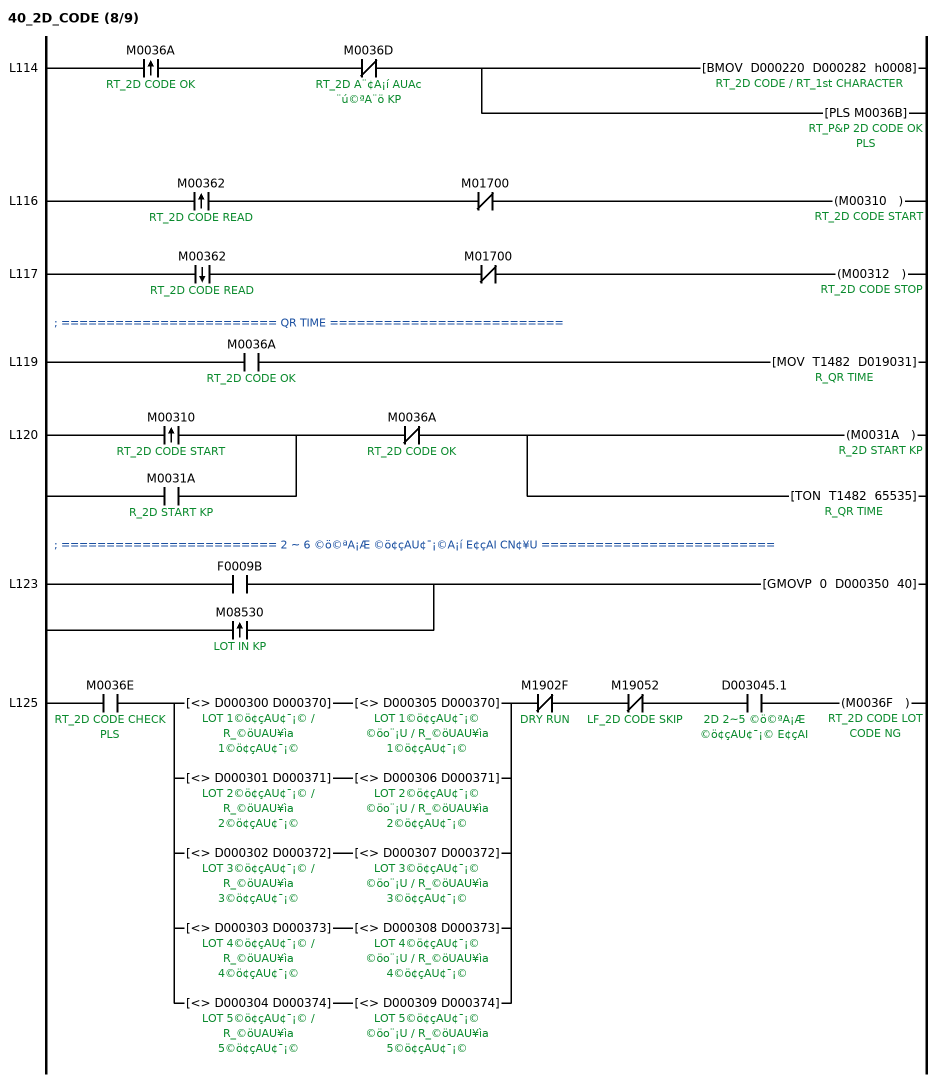
[picture p240: 40_2D_CODE rungs L114-L125]
; L114
LOADP     M0036A	// RT_2D CODE OK
AND NOT   M0036D	// RT_2D A¨¢A¡í AUAc ¨ú©ªA¨ö KP
BMOV      D000220 D000282 h0008	// RT_2D CODE / RT_1st CHARACTER
OUTP      M0036B	// RT_P&P 2D CODE OK PLS
; L116
LOADP     M00362	// RT_2D CODE READ
AND NOT   M01700
OUT       M00310	// RT_2D CODE START
; L117
LOADN     M00362	// RT_2D CODE READ
AND NOT   M01700
OUT       M00312	// RT_2D CODE STOP
// ======================== QR TIME ==========================
; L119
LOAD      M0036A	// RT_2D CODE OK
MOV       T1482 D019031	// R_QR TIME
; L120
LOADP     M00310	// RT_2D CODE START
OR        M0031A	// R_2D START KP
AND NOT   M0036A	// RT_2D CODE OK
OUT       M0031A	// R_2D START KP
TON       T1482 65535	// R_QR TIME
// ======================== 2 ~ 6 ©ö©ªA¡Æ ©ö¢çAU¢¯¡©A¡í E¢çAI CN¢¥U ==========================
; L123
LOAD      F0009B
ORP       M08530	// LOT IN KP
GMOVP     0 D000350 40
; L125
LOAD      M0036E	// RT_2D CODE CHECK PLS
LOAD<>    D000300 D000370	// LOT 1©ö¢çAU¢¯¡© / R_©öUAU¥ìa 1©ö¢çAU¢¯¡©
AND<>     D000305 D000370	// LOT 1©ö¢çAU¢¯¡© ©öo¨¡U / R_©öUAU¥ìa 1©ö¢çAU¢¯¡©
LOAD<>    D000301 D000371	// LOT 2©ö¢çAU¢¯¡© / R_©öUAU¥ìa 2©ö¢çAU¢¯¡©
AND<>     D000306 D000371	// LOT 2©ö¢çAU¢¯¡© ©öo¨¡U / R_©öUAU¥ìa 2©ö¢çAU¢¯¡©
OR LOAD
LOAD<>    D000302 D000372	// LOT 3©ö¢çAU¢¯¡© / R_©öUAU¥ìa 3©ö¢çAU¢¯¡©
AND<>     D000307 D000372	// LOT 3©ö¢çAU¢¯¡© ©öo¨¡U / R_©öUAU¥ìa 3©ö¢çAU¢¯¡©
OR LOAD
LOAD<>    D000303 D000373	// LOT 4©ö¢çAU¢¯¡© / R_©öUAU¥ìa 4©ö¢çAU¢¯¡©
AND<>     D000308 D000373	// LOT 4©ö¢çAU¢¯¡© ©öo¨¡U / R_©öUAU¥ìa 4©ö¢çAU¢¯¡©
OR LOAD
LOAD<>    D000304 D000374	// LOT 5©ö¢çAU¢¯¡© / R_©öUAU¥ìa 5©ö¢çAU¢¯¡©
AND<>     D000309 D000374	// LOT 5©ö¢çAU¢¯¡© ©öo¨¡U / R_©öUAU¥ìa 5©ö¢çAU¢¯¡©
OR LOAD
AND LOAD
AND NOT   M1902F	// DRY RUN
AND NOT   M19052	// LF_2D CODE SKIP
AND       D003045.1	// 2D 2~5 ©ö©ªA¡Æ ©ö¢çAU¢¯¡© E¢çAI
OUT       M0036F	// RT_2D CODE LOT CODE NG

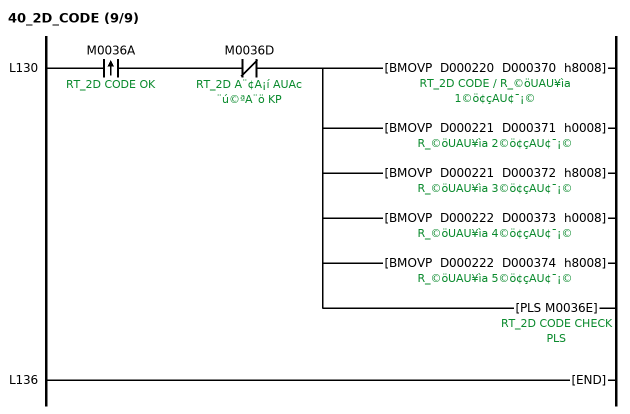
; L130
LOADP     M0036A	// RT_2D CODE OK
AND NOT   M0036D	// RT_2D A¨¢A¡í AUAc ¨ú©ªA¨ö KP
BMOVP     D000220 D000370 h8008	// RT_2D CODE / R_©öUAU¥ìa 1©ö¢çAU¢¯¡©
BMOVP     D000221 D000371 h0008	// R_©öUAU¥ìa 2©ö¢çAU¢¯¡©
BMOVP     D000221 D000372 h8008	// R_©öUAU¥ìa 3©ö¢çAU¢¯¡©
BMOVP     D000222 D000373 h0008	// R_©öUAU¥ìa 4©ö¢çAU¢¯¡©
BMOVP     D000222 D000374 h8008	// R_©öUAU¥ìa 5©ö¢çAU¢¯¡©
OUTP      M0036E	// RT_2D CODE CHECK PLS
; L136
END

PROGRAM 41_MES (task: ¨ö¨¬A¥ì CA¡¤I¡¾¡¿¡¤¡Í)

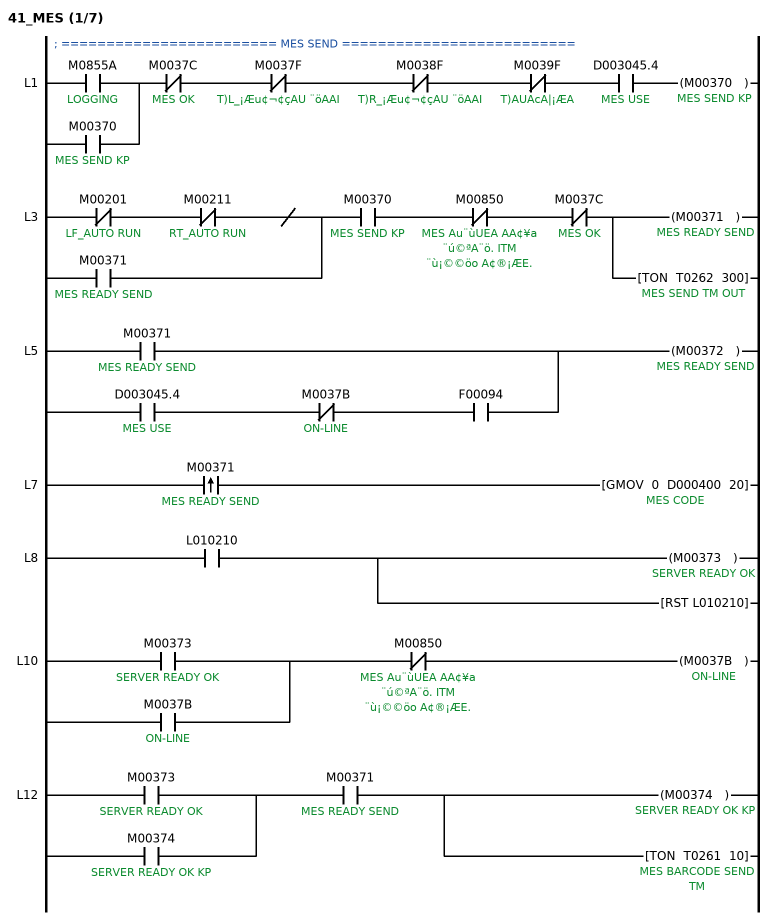
// ======================== MES SEND ==========================
; L1
LOAD      M0855A	// LOGGING
OR        M00370	// MES SEND KP
AND NOT   M0037C	// MES OK
AND NOT   M0037F	// T)L_¡Æu¢¬¢çAU ¨öAAI
AND NOT   M0038F	// T)R_¡Æu¢¬¢çAU ¨öAAI
AND NOT   M0039F	// T)AUAcA|¡ÆA
AND       D003045.4	// MES USE
OUT       M00370	// MES SEND KP
; L3
LOAD NOT  M00201	// LF_AUTO RUN
AND NOT   M00211	// RT_AUTO RUN
NOT
OR        M00371	// MES READY SEND
AND       M00370	// MES SEND KP
AND NOT   M00850	// MES Au¨ùUEA AA¢¥a ¨ú©ªA¨ö. ITM ¨ù¡©©öo A¢®¡ÆE.
AND NOT   M0037C	// MES OK
OUT       M00371	// MES READY SEND
TON       T0262 300	// MES SEND TM OUT
; L5
LOAD      M00371	// MES READY SEND
LOAD      D003045.4	// MES USE
AND NOT   M0037B	// ON-LINE
AND       F00094
OR LOAD
OUT       M00372	// MES READY SEND
; L7
LOADP     M00371	// MES READY SEND
GMOV      0 D000400 20	// MES CODE
; L8
LOAD      L010210
OUT       M00373	// SERVER READY OK
RST       L010210
; L10
LOAD      M00373	// SERVER READY OK
OR        M0037B	// ON-LINE
AND NOT   M00850	// MES Au¨ùUEA AA¢¥a ¨ú©ªA¨ö. ITM ¨ù¡©©öo A¢®¡ÆE.
OUT       M0037B	// ON-LINE
; L12
LOAD      M00373	// SERVER READY OK
OR        M00374	// SERVER READY OK KP
AND       M00371	// MES READY SEND
OUT       M00374	// SERVER READY OK KP
TON       T0261 10	// MES BARCODE SEND TM

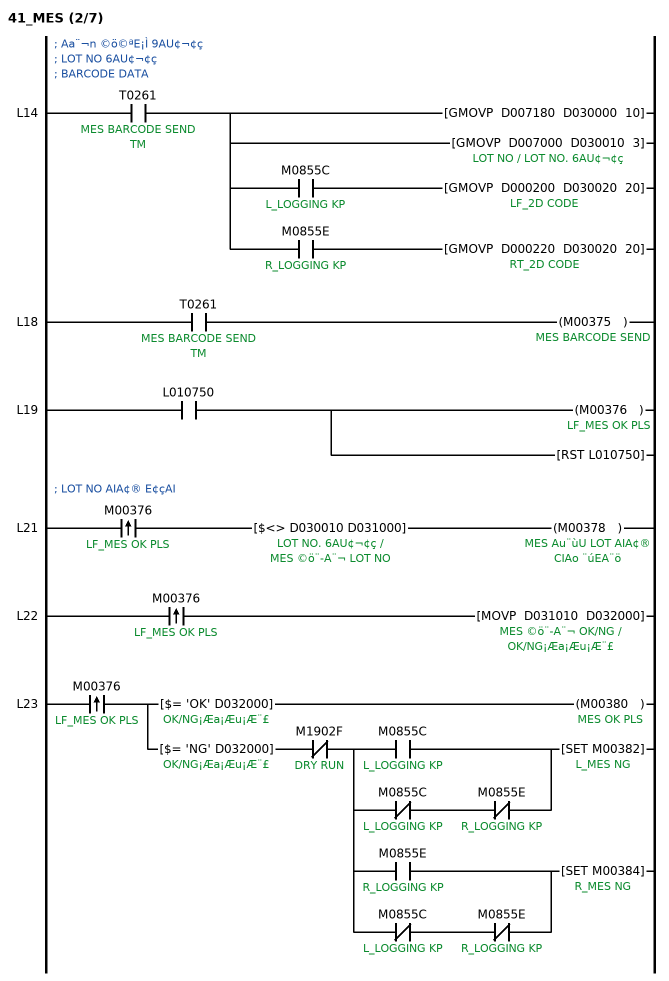
; L14
LOAD      T0261	// MES BARCODE SEND TM
GMOVP     D007180 D030000 10
GMOVP     D007000 D030010 3	// LOT NO / LOT NO. 6AU¢¬¢ç
MPUSH
AND       M0855C	// L_LOGGING KP
GMOVP     D000200 D030020 20	// LF_2D CODE
MPOP
AND       M0855E	// R_LOGGING KP
GMOVP     D000220 D030020 20	// RT_2D CODE
// output comment: Aa¨¬n ©ö©ªE¡Ì 9AU¢¬¢ç
// output comment: LOT NO 6AU¢¬¢ç
// output comment: BARCODE DATA
; L18
LOAD      T0261	// MES BARCODE SEND TM
OUT       M00375	// MES BARCODE SEND
; L19
LOAD      L010750
OUT       M00376	// LF_MES OK PLS
RST       L010750
; L21
LOADP     M00376	// LF_MES OK PLS
AND$<>    D030010 D031000	// LOT NO. 6AU¢¬¢ç / MES ©ö¨­A¨¬ LOT NO
OUT       M00378	// MES Au¨ùU LOT AIA¢® CIAo ¨úEA¨ö
// output comment: LOT NO AIA¢® E¢çAI
; L22
LOADP     M00376	// LF_MES OK PLS
MOVP      D031010 D032000	// MES ©ö¨­A¨¬ OK/NG / OK/NG¡Æa¡Æu¡Æ¨£
; L23
LOADP     M00376	// LF_MES OK PLS
MPUSH
AND$=     'OK' D032000	// OK/NG¡Æa¡Æu¡Æ¨£
OUT       M00380	// MES OK PLS
MPOP
AND$=     'NG' D032000	// OK/NG¡Æa¡Æu¡Æ¨£
AND NOT   M1902F	// DRY RUN
MPUSH
LOAD      M0855C	// L_LOGGING KP
LOAD NOT  M0855C	// L_LOGGING KP
AND NOT   M0855E	// R_LOGGING KP
OR LOAD
AND LOAD
SET       M00382	// L_MES NG
MPOP
LOAD      M0855E	// R_LOGGING KP
LOAD NOT  M0855C	// L_LOGGING KP
AND NOT   M0855E	// R_LOGGING KP
OR LOAD
AND LOAD
SET       M00384	// R_MES NG

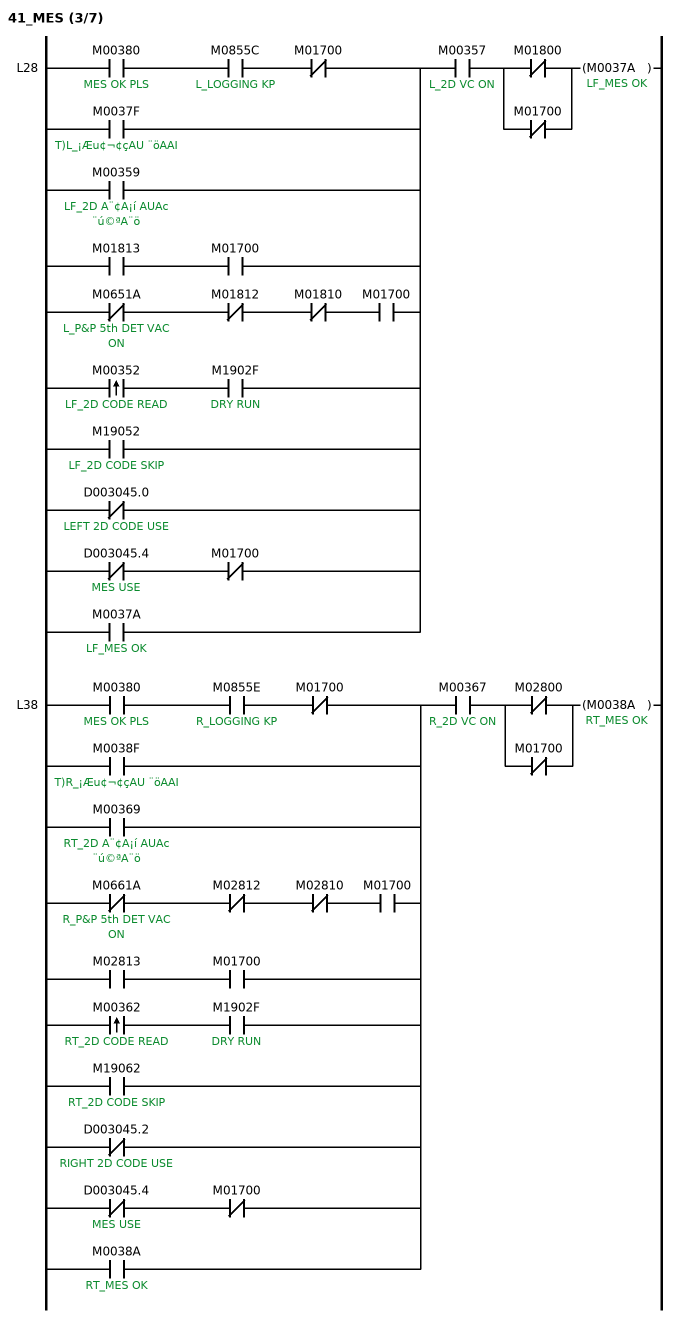
; L28
LOAD      M00380	// MES OK PLS
AND       M0855C	// L_LOGGING KP
AND NOT   M01700
OR        M0037F	// T)L_¡Æu¢¬¢çAU ¨öAAI
OR        M00359	// LF_2D A¨¢A¡í AUAc ¨ú©ªA¨ö
LOAD      M01813
AND       M01700
OR LOAD
LOAD NOT  M0651A	// L_P&P 5th DET VAC ON
AND NOT   M01812
AND NOT   M01810
AND       M01700
OR LOAD
LOADP     M00352	// LF_2D CODE READ
AND       M1902F	// DRY RUN
OR LOAD
OR        M19052	// LF_2D CODE SKIP
OR NOT    D003045.0	// LEFT 2D CODE USE
LOAD NOT  D003045.4	// MES USE
AND NOT   M01700
OR LOAD
OR        M0037A	// LF_MES OK
AND       M00357	// L_2D VC ON
LOAD NOT  M01800
OR NOT    M01700
AND LOAD
OUT       M0037A	// LF_MES OK
; L38
LOAD      M00380	// MES OK PLS
AND       M0855E	// R_LOGGING KP
AND NOT   M01700
OR        M0038F	// T)R_¡Æu¢¬¢çAU ¨öAAI
OR        M00369	// RT_2D A¨¢A¡í AUAc ¨ú©ªA¨ö
LOAD NOT  M0661A	// R_P&P 5th DET VAC ON
AND NOT   M02812
AND NOT   M02810
AND       M01700
OR LOAD
LOAD      M02813
AND       M01700
OR LOAD
LOADP     M00362	// RT_2D CODE READ
AND       M1902F	// DRY RUN
OR LOAD
OR        M19062	// RT_2D CODE SKIP
OR NOT    D003045.2	// RIGHT 2D CODE USE
LOAD NOT  D003045.4	// MES USE
AND NOT   M01700
OR LOAD
OR        M0038A	// RT_MES OK
AND       M00367	// R_2D VC ON
LOAD NOT  M02800
OR NOT    M01700
AND LOAD
OUT       M0038A	// RT_MES OK

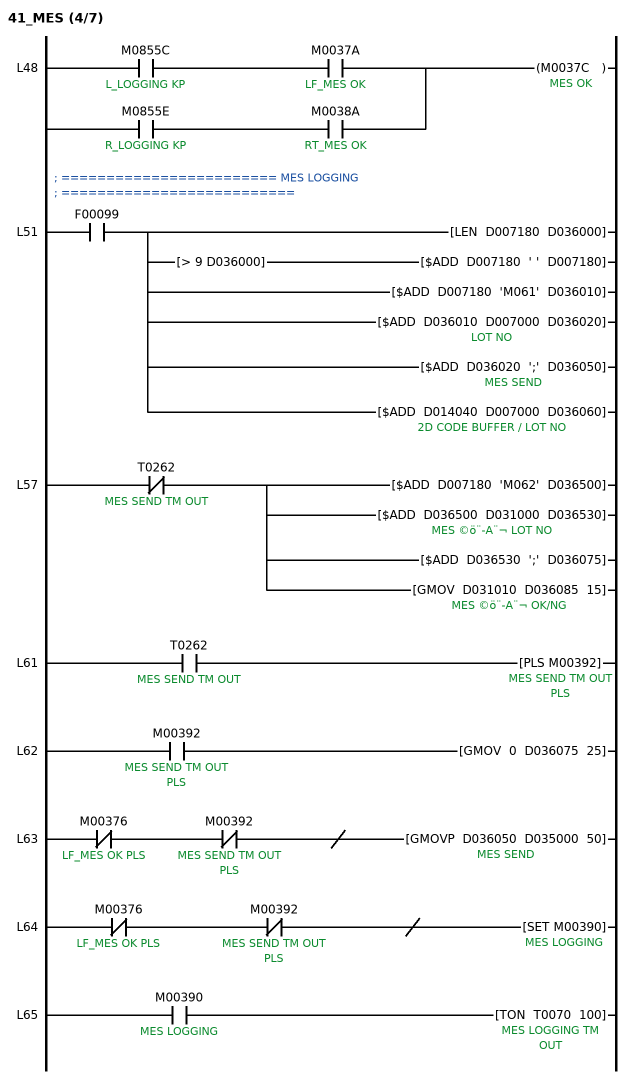
; L48
LOAD      M0855C	// L_LOGGING KP
AND       M0037A	// LF_MES OK
LOAD      M0855E	// R_LOGGING KP
AND       M0038A	// RT_MES OK
OR LOAD
OUT       M0037C	// MES OK
// ======================== MES LOGGING ==========================
; L51
LOAD      F00099
LEN       D007180 D036000
MPUSH
AND>      9 D036000
$ADD      D007180 ' ' D007180
MPOP
$ADD      D007180 'M061' D036010
$ADD      D036010 D007000 D036020	// LOT NO
$ADD      D036020 ';' D036050	// MES SEND
$ADD      D014040 D007000 D036060	// 2D CODE BUFFER / LOT NO
; L57
LOAD NOT  T0262	// MES SEND TM OUT
$ADD      D007180 'M062' D036500
$ADD      D036500 D031000 D036530	// MES ©ö¨­A¨¬ LOT NO
$ADD      D036530 ';' D036075
GMOV      D031010 D036085 15	// MES ©ö¨­A¨¬ OK/NG
; L61
LOAD      T0262	// MES SEND TM OUT
OUTP      M00392	// MES SEND TM OUT PLS
; L62
LOAD      M00392	// MES SEND TM OUT PLS
GMOV      0 D036075 25
; L63
LOAD NOT  M00376	// LF_MES OK PLS
AND NOT   M00392	// MES SEND TM OUT PLS
NOT
GMOVP     D036050 D035000 50	// MES SEND
; L64
LOAD NOT  M00376	// LF_MES OK PLS
AND NOT   M00392	// MES SEND TM OUT PLS
NOT
SET       M00390	// MES LOGGING
; L65
LOAD      M00390	// MES LOGGING
TON       T0070 100	// MES LOGGING TM OUT

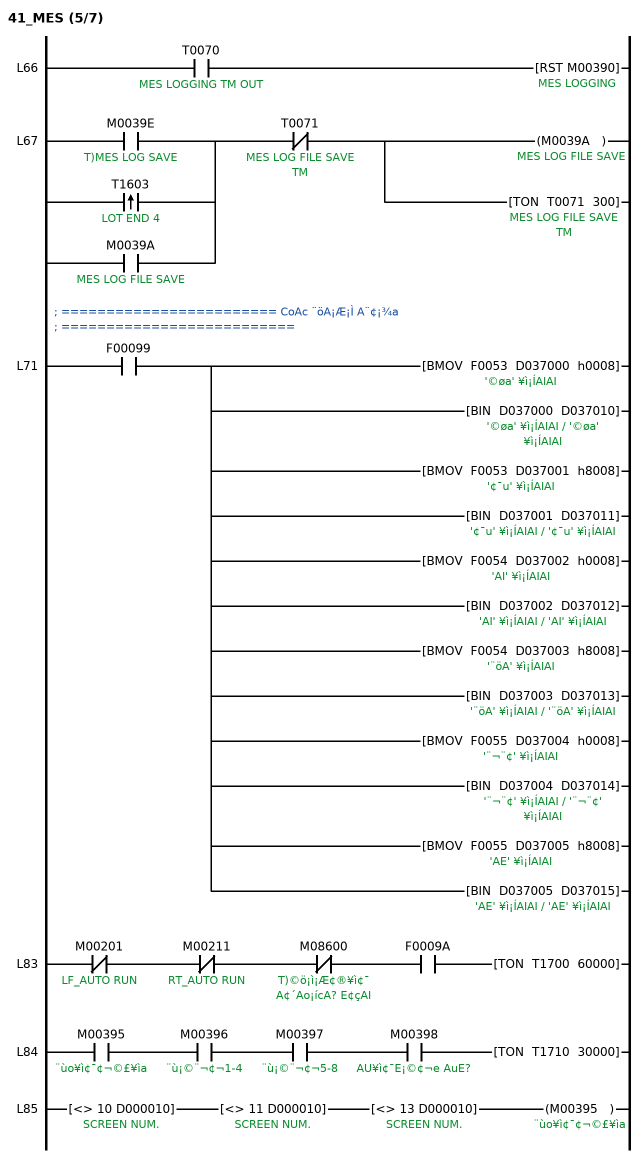
; L66
LOAD      T0070	// MES LOGGING TM OUT
RST       M00390	// MES LOGGING
; L67
LOAD      M0039E	// T)MES LOG SAVE
ORP       T1603	// LOT END 4
OR        M0039A	// MES LOG FILE SAVE
AND NOT   T0071	// MES LOG FILE SAVE TM
OUT       M0039A	// MES LOG FILE SAVE
TON       T0071 300	// MES LOG FILE SAVE TM
// ======================== CoAc ¨öA¡Æ¡Ì A¨¢¡¾a ==========================
; L71
LOAD      F00099
BMOV      F0053 D037000 h0008	// '©øa' ¥ì¡ÍAIAI
BIN       D037000 D037010	// '©øa' ¥ì¡ÍAIAI / '©øa' ¥ì¡ÍAIAI
BMOV      F0053 D037001 h8008	// '¢¯u' ¥ì¡ÍAIAI
BIN       D037001 D037011	// '¢¯u' ¥ì¡ÍAIAI / '¢¯u' ¥ì¡ÍAIAI
BMOV      F0054 D037002 h0008	// 'AI' ¥ì¡ÍAIAI
BIN       D037002 D037012	// 'AI' ¥ì¡ÍAIAI / 'AI' ¥ì¡ÍAIAI
BMOV      F0054 D037003 h8008	// '¨öA' ¥ì¡ÍAIAI
BIN       D037003 D037013	// '¨öA' ¥ì¡ÍAIAI / '¨öA' ¥ì¡ÍAIAI
BMOV      F0055 D037004 h0008	// '¨¬¨¢' ¥ì¡ÍAIAI
BIN       D037004 D037014	// '¨¬¨¢' ¥ì¡ÍAIAI / '¨¬¨¢' ¥ì¡ÍAIAI
BMOV      F0055 D037005 h8008	// 'AE' ¥ì¡ÍAIAI
BIN       D037005 D037015	// 'AE' ¥ì¡ÍAIAI / 'AE' ¥ì¡ÍAIAI
; L83
LOAD NOT  M00201	// LF_AUTO RUN
AND NOT   M00211	// RT_AUTO RUN
AND NOT   M08600	// T)©ö¡ì¡Æ¢®¥ì¢¯ A¢´Ao¡ícA? E¢çAI
AND       F0009A
TON       T1700 60000
; L84
LOAD      M00395	// ¨ùo¥ì¢¯¢¬©£¥ìa
AND       M00396	// ¨ù¡©¨¬¢¬1-4
AND       M00397	// ¨ù¡©¨¬¢¬5-8
AND       M00398	// AU¥ì¢¯E¡©¢¬e AuE?
TON       T1710 30000
; L85
LOAD<>    10 D000010	// SCREEN NUM.
AND<>     11 D000010	// SCREEN NUM.
AND<>     13 D000010	// SCREEN NUM.
OUT       M00395	// ¨ùo¥ì¢¯¢¬©£¥ìa

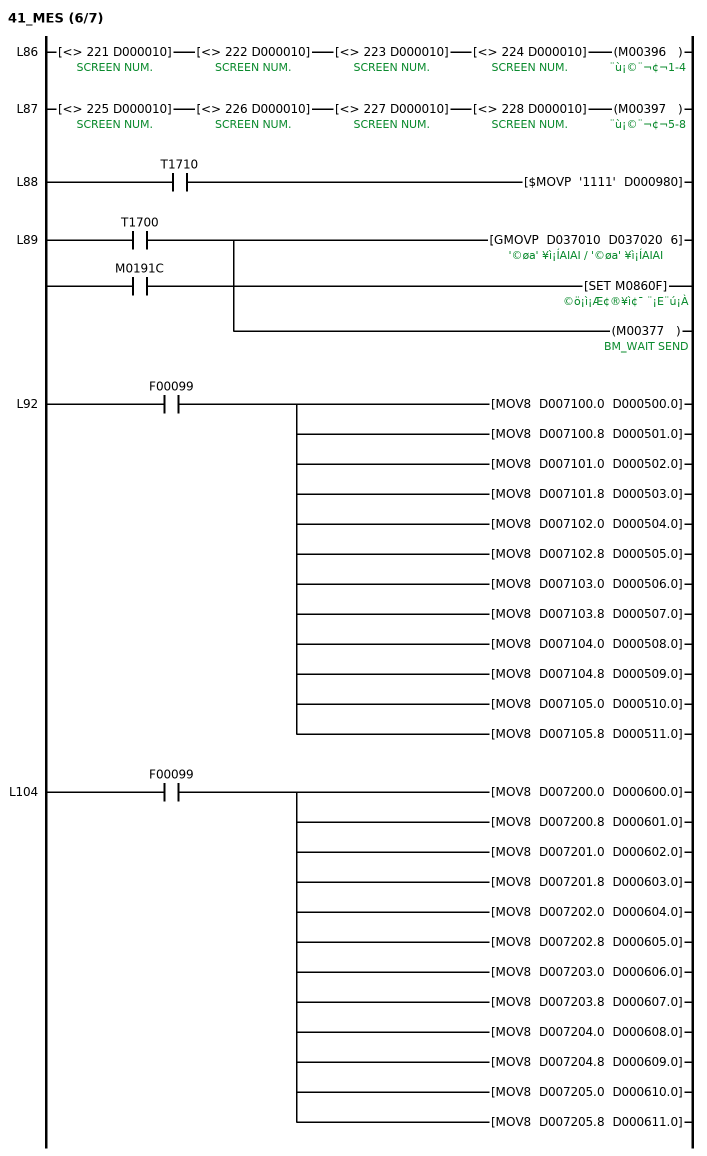
; L86
LOAD<>    221 D000010	// SCREEN NUM.
AND<>     222 D000010	// SCREEN NUM.
AND<>     223 D000010	// SCREEN NUM.
AND<>     224 D000010	// SCREEN NUM.
OUT       M00396	// ¨ù¡©¨¬¢¬1-4
; L87
LOAD<>    225 D000010	// SCREEN NUM.
AND<>     226 D000010	// SCREEN NUM.
AND<>     227 D000010	// SCREEN NUM.
AND<>     228 D000010	// SCREEN NUM.
OUT       M00397	// ¨ù¡©¨¬¢¬5-8
; L88
LOAD      T1710
$MOVP     '1111' D000980
; L89
LOAD      T1700
OR        M0191C
GMOVP     D037010 D037020 6	// '©øa' ¥ì¡ÍAIAI / '©øa' ¥ì¡ÍAIAI
SET       M0860F	// ©ö¡ì¡Æ¢®¥ì¢¯ ¨¡E¨ú¡À
OUT       M00377	// BM_WAIT SEND
; L92
LOAD      F00099
MOV8      D007100.0 D000500.0
MOV8      D007100.8 D000501.0
MOV8      D007101.0 D000502.0
MOV8      D007101.8 D000503.0
MOV8      D007102.0 D000504.0
MOV8      D007102.8 D000505.0
MOV8      D007103.0 D000506.0
MOV8      D007103.8 D000507.0
MOV8      D007104.0 D000508.0
MOV8      D007104.8 D000509.0
MOV8      D007105.0 D000510.0
MOV8      D007105.8 D000511.0
; L104
LOAD      F00099
MOV8      D007200.0 D000600.0
MOV8      D007200.8 D000601.0
MOV8      D007201.0 D000602.0
MOV8      D007201.8 D000603.0
MOV8      D007202.0 D000604.0
MOV8      D007202.8 D000605.0
MOV8      D007203.0 D000606.0
MOV8      D007203.8 D000607.0
MOV8      D007204.0 D000608.0
MOV8      D007204.8 D000609.0
MOV8      D007205.0 D000610.0
MOV8      D007205.8 D000611.0

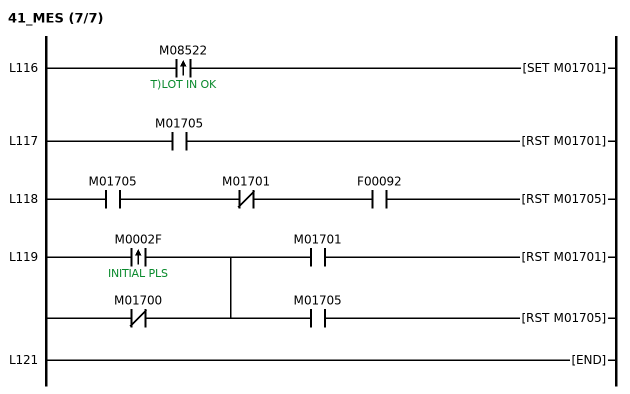
; L116
LOADP     M08522	// T)LOT IN OK
SET       M01701
; L117
LOAD      M01705
RST       M01701
; L118
LOAD      M01705
AND NOT   M01701
AND       F00092
RST       M01705
; L119
LOADP     M0002F	// INITIAL PLS
OR NOT    M01700
MPUSH
AND       M01701
RST       M01701
MPOP
AND       M01705
RST       M01705
; L121
END

PROGRAM 51_MT_01_2_3_4 (task: ¨ö¨¬A¥ì CA¡¤I¡¾¡¿¡¤¡Í)

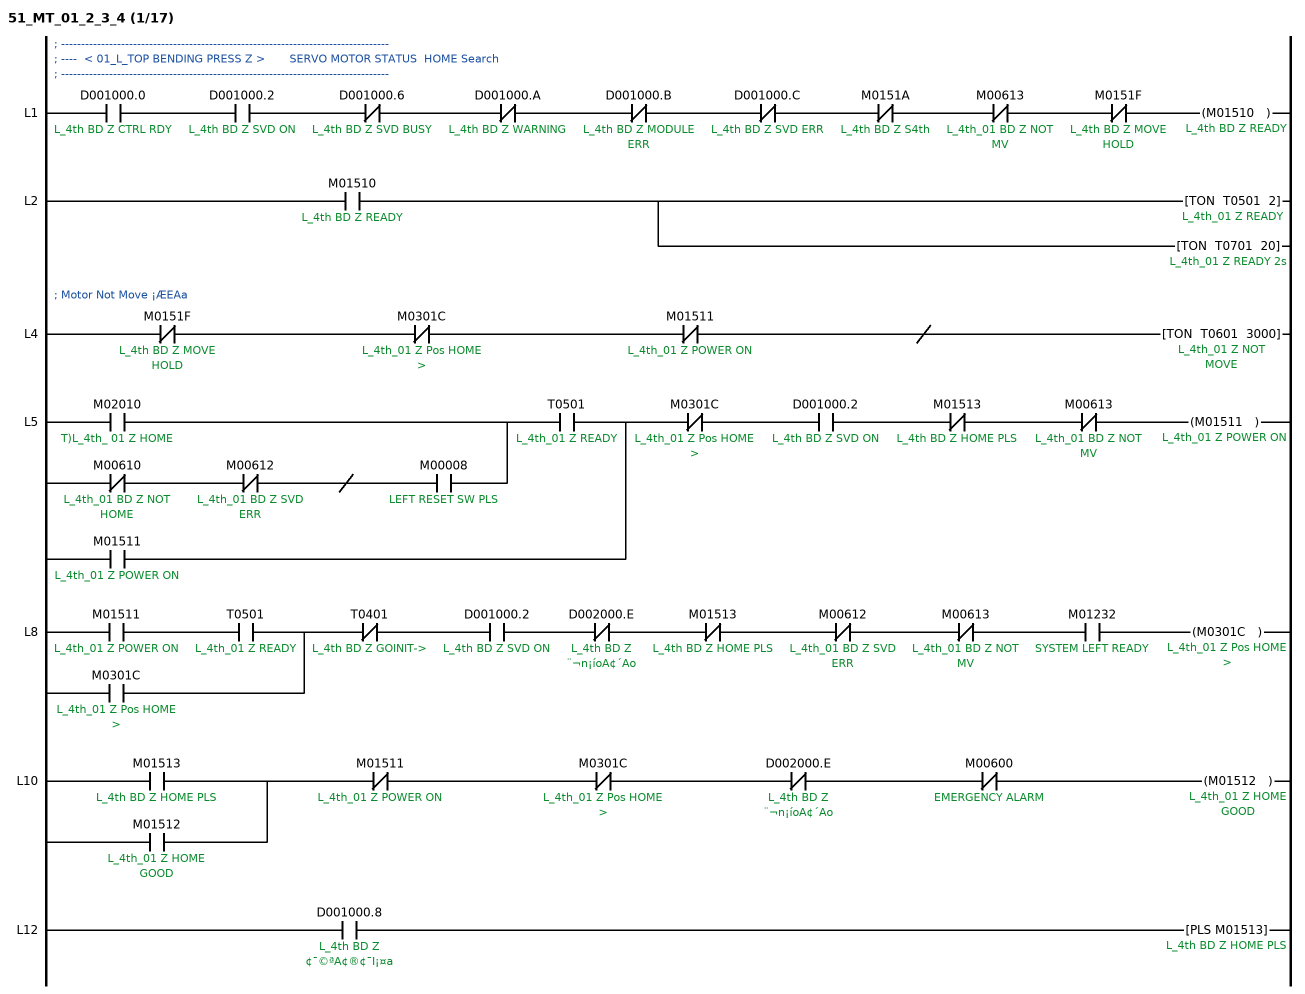
// ----------------------------------------------------------------------------------
// 
// ----  < 01_L_TOP BENDING PRESS Z >       SERVO MOTOR STATUS  HOME Search
// 
// ----------------------------------------------------------------------------------
; L1
LOAD      D001000.0	// L_4th BD Z CTRL RDY
AND       D001000.2	// L_4th BD Z SVD ON
AND NOT   D001000.6	// L_4th BD Z SVD BUSY
AND NOT   D001000.A	// L_4th BD Z WARNING
AND NOT   D001000.B	// L_4th BD Z MODULE ERR
AND NOT   D001000.C	// L_4th BD Z SVD ERR
AND NOT   M0151A	// L_4th BD Z S4th
AND NOT   M00613	// L_4th_01 BD Z NOT MV
AND NOT   M0151F	// L_4th BD Z MOVE HOLD
OUT       M01510	// L_4th BD Z READY
; L2
LOAD      M01510	// L_4th BD Z READY
TON       T0501 2	// L_4th_01 Z READY
TON       T0701 20	// L_4th_01 Z READY 2s
; L4
LOAD NOT  M0151F	// L_4th BD Z MOVE HOLD
AND NOT   M0301C	// L_4th_01 Z Pos HOME >
AND NOT   M01511	// L_4th_01 Z POWER ON
NOT
TON       T0601 3000	// L_4th_01 Z NOT MOVE
// output comment: Motor Not Move ¡ÆEAa
; L5
LOAD      M02010	// T)L_4th_ 01 Z HOME
LOAD NOT  M00610	// L_4th_01 BD Z NOT HOME
AND NOT   M00612	// L_4th_01 BD Z SVD ERR
NOT
AND       M00008	// LEFT RESET SW PLS
OR LOAD
AND       T0501	// L_4th_01 Z READY
OR        M01511	// L_4th_01 Z POWER ON
AND NOT   M0301C	// L_4th_01 Z Pos HOME >
AND       D001000.2	// L_4th BD Z SVD ON
AND NOT   M01513	// L_4th BD Z HOME PLS
AND NOT   M00613	// L_4th_01 BD Z NOT MV
OUT       M01511	// L_4th_01 Z POWER ON
; L8
LOAD      M01511	// L_4th_01 Z POWER ON
AND       T0501	// L_4th_01 Z READY
OR        M0301C	// L_4th_01 Z Pos HOME >
AND NOT   T0401	// L_4th BD Z GOINIT->
AND       D001000.2	// L_4th BD Z SVD ON
AND NOT   D002000.E	// L_4th BD Z ¨¬n¡íoA¢´Ao
AND NOT   M01513	// L_4th BD Z HOME PLS
AND NOT   M00612	// L_4th_01 BD Z SVD ERR
AND NOT   M00613	// L_4th_01 BD Z NOT MV
AND       M01232	// SYSTEM LEFT READY
OUT       M0301C	// L_4th_01 Z Pos HOME >
; L10
LOAD      M01513	// L_4th BD Z HOME PLS
OR        M01512	// L_4th_01 Z HOME GOOD
AND NOT   M01511	// L_4th_01 Z POWER ON
AND NOT   M0301C	// L_4th_01 Z Pos HOME >
AND NOT   D002000.E	// L_4th BD Z ¨¬n¡íoA¢´Ao
AND NOT   M00600	// EMERGENCY ALARM
OUT       M01512	// L_4th_01 Z HOME GOOD
; L12
LOAD      D001000.8	// L_4th BD Z ¢¯©ªA¢®¢¯I¡¤a
OUTP      M01513	// L_4th BD Z HOME PLS

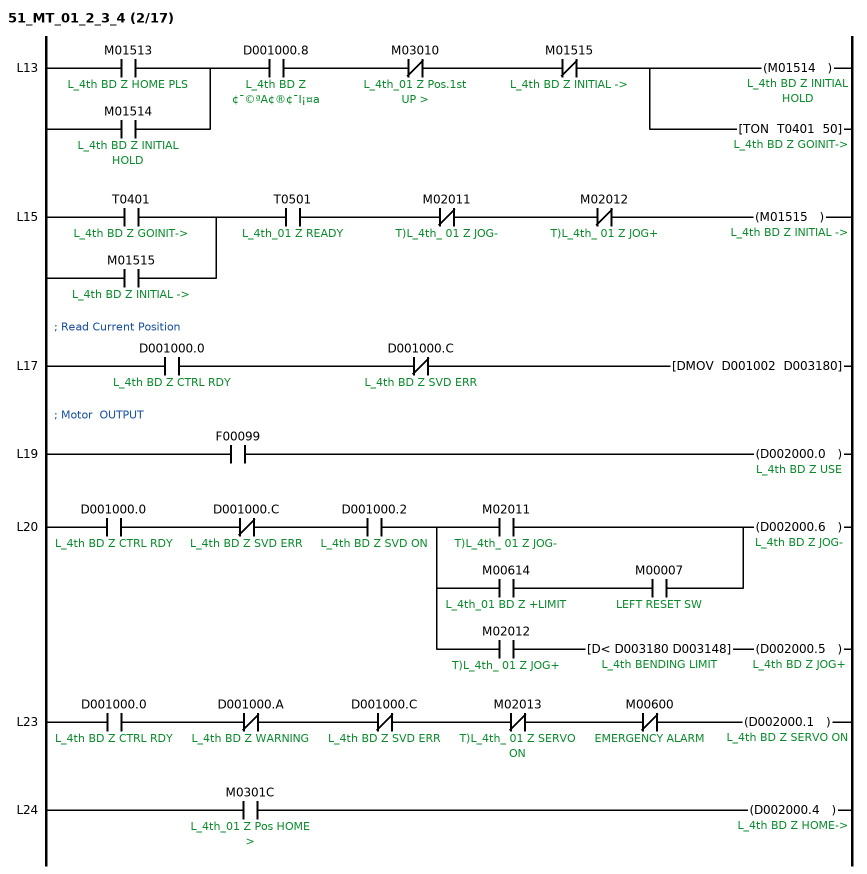
; L13
LOAD      M01513	// L_4th BD Z HOME PLS
OR        M01514	// L_4th BD Z INITIAL HOLD
AND       D001000.8	// L_4th BD Z ¢¯©ªA¢®¢¯I¡¤a
AND NOT   M03010	// L_4th_01 Z Pos.1st     UP >
AND NOT   M01515	// L_4th BD Z INITIAL ->
OUT       M01514	// L_4th BD Z INITIAL HOLD
TON       T0401 50	// L_4th BD Z GOINIT->
; L15
LOAD      T0401	// L_4th BD Z GOINIT->
OR        M01515	// L_4th BD Z INITIAL ->
AND       T0501	// L_4th_01 Z READY
AND NOT   M02011	// T)L_4th_ 01 Z JOG-
AND NOT   M02012	// T)L_4th_ 01 Z JOG+
OUT       M01515	// L_4th BD Z INITIAL ->
; L17
LOAD      D001000.0	// L_4th BD Z CTRL RDY
AND NOT   D001000.C	// L_4th BD Z SVD ERR
DMOV      D001002 D003180
// output comment: Read Current Position
//  Motor  OUTPUT
; L19
LOAD      F00099
OUT       D002000.0	// L_4th BD Z USE
; L20
LOAD      D001000.0	// L_4th BD Z CTRL RDY
AND NOT   D001000.C	// L_4th BD Z SVD ERR
AND       D001000.2	// L_4th BD Z SVD ON
MPUSH
LOAD      M02011	// T)L_4th_ 01 Z JOG-
LOAD      M00614	// L_4th_01 BD Z +LIMIT
AND       M00007	// LEFT RESET SW
OR LOAD
AND LOAD
OUT       D002000.6	// L_4th BD Z JOG-
MPOP
AND       M02012	// T)L_4th_ 01 Z JOG+
ANDD<     D003180 D003148	// L_4th BENDING LIMIT
OUT       D002000.5	// L_4th BD Z JOG+
; L23
LOAD      D001000.0	// L_4th BD Z CTRL RDY
AND NOT   D001000.A	// L_4th BD Z WARNING
AND NOT   D001000.C	// L_4th BD Z SVD ERR
AND NOT   M02013	// T)L_4th_ 01 Z SERVO ON
AND NOT   M00600	// EMERGENCY ALARM
OUT       D002000.1	// L_4th BD Z SERVO ON
; L24
LOAD      M0301C	// L_4th_01 Z Pos HOME >
OUT       D002000.4	// L_4th BD Z HOME->

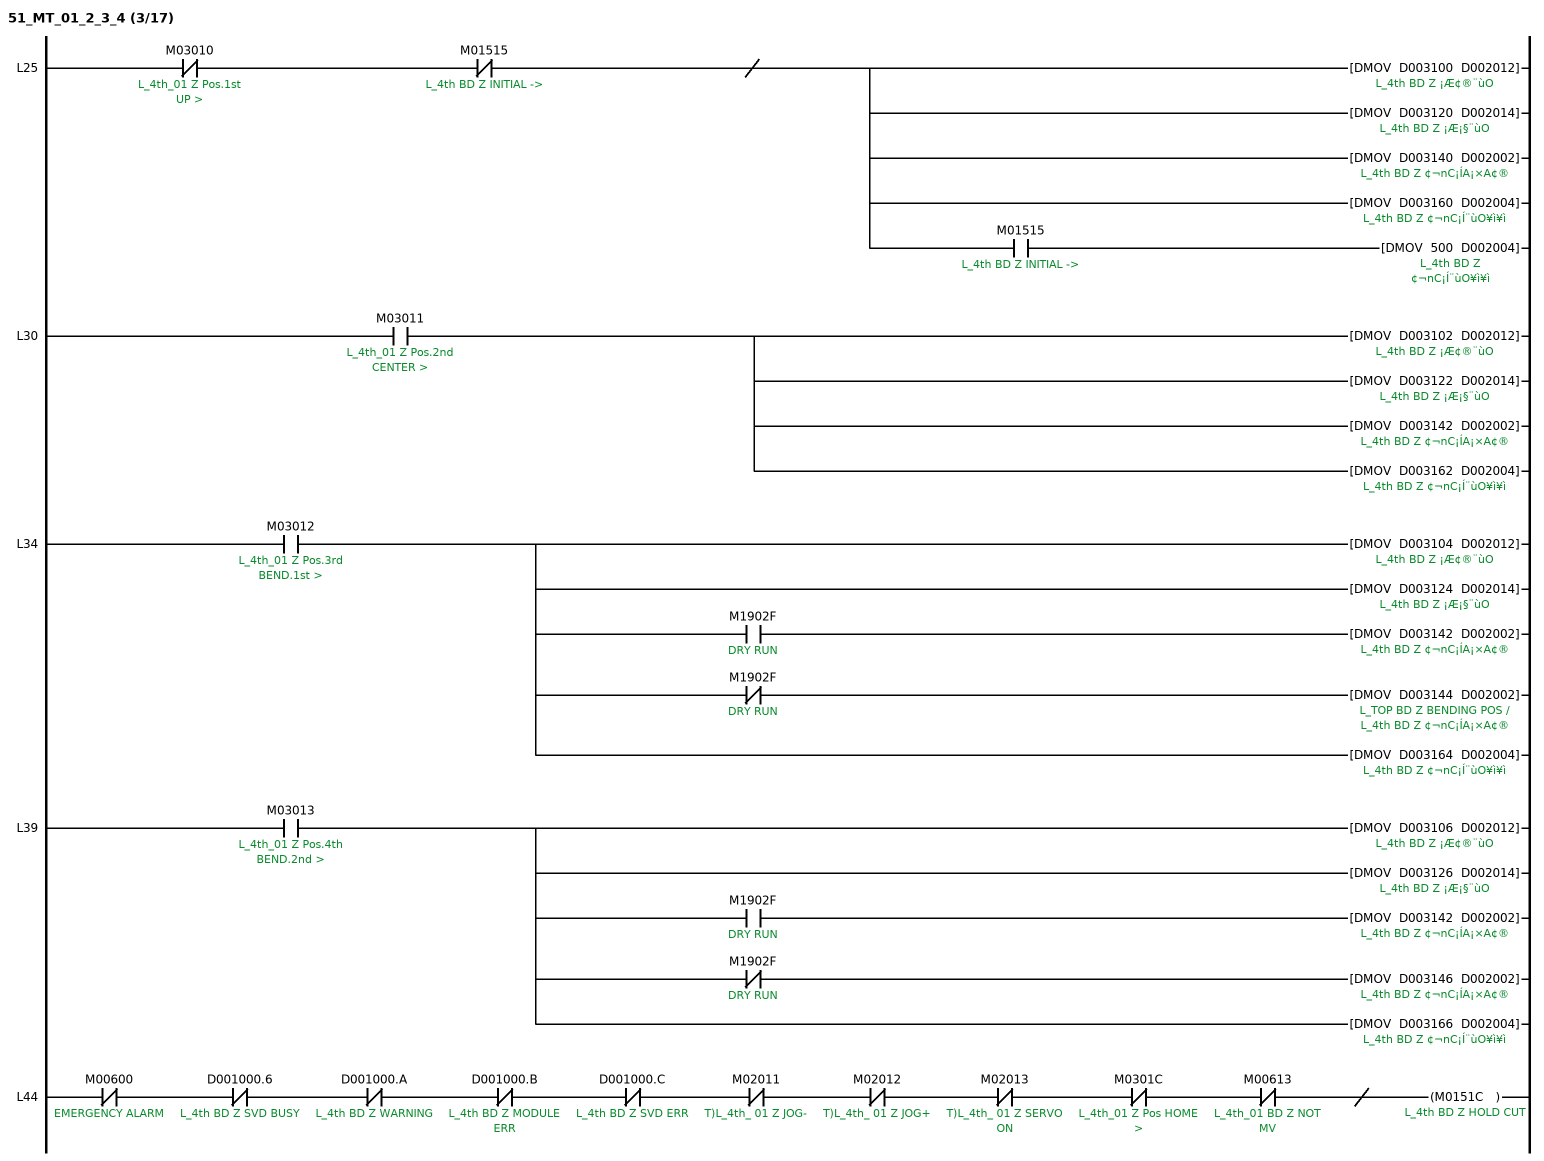
; L25
LOAD NOT  M03010	// L_4th_01 Z Pos.1st     UP >
AND NOT   M01515	// L_4th BD Z INITIAL ->
NOT
DMOV      D003100 D002012	// L_4th BD Z ¡Æ¢®¨ùO
DMOV      D003120 D002014	// L_4th BD Z ¡Æ¡§¨ùO
DMOV      D003140 D002002	// L_4th BD Z ¢¬nC¡ÍA¡×A¢®
DMOV      D003160 D002004	// L_4th BD Z ¢¬nC¡Í¨ùO¥ì¥ì
AND       M01515	// L_4th BD Z INITIAL ->
DMOV      500 D002004	// L_4th BD Z ¢¬nC¡Í¨ùO¥ì¥ì
; L30
LOAD      M03011	// L_4th_01 Z Pos.2nd CENTER >
DMOV      D003102 D002012	// L_4th BD Z ¡Æ¢®¨ùO
DMOV      D003122 D002014	// L_4th BD Z ¡Æ¡§¨ùO
DMOV      D003142 D002002	// L_4th BD Z ¢¬nC¡ÍA¡×A¢®
DMOV      D003162 D002004	// L_4th BD Z ¢¬nC¡Í¨ùO¥ì¥ì
; L34
LOAD      M03012	// L_4th_01 Z Pos.3rd BEND.1st >
DMOV      D003104 D002012	// L_4th BD Z ¡Æ¢®¨ùO
DMOV      D003124 D002014	// L_4th BD Z ¡Æ¡§¨ùO
MPUSH
AND       M1902F	// DRY RUN
DMOV      D003142 D002002	// L_4th BD Z ¢¬nC¡ÍA¡×A¢®
MLOAD
AND NOT   M1902F	// DRY RUN
DMOV      D003144 D002002	// L_TOP BD Z BENDING POS / L_4th BD Z ¢¬nC¡ÍA¡×A¢®
MPOP
DMOV      D003164 D002004	// L_4th BD Z ¢¬nC¡Í¨ùO¥ì¥ì
; L39
LOAD      M03013	// L_4th_01 Z Pos.4th BEND.2nd >
DMOV      D003106 D002012	// L_4th BD Z ¡Æ¢®¨ùO
DMOV      D003126 D002014	// L_4th BD Z ¡Æ¡§¨ùO
MPUSH
AND       M1902F	// DRY RUN
DMOV      D003142 D002002	// L_4th BD Z ¢¬nC¡ÍA¡×A¢®
MLOAD
AND NOT   M1902F	// DRY RUN
DMOV      D003146 D002002	// L_4th BD Z ¢¬nC¡ÍA¡×A¢®
MPOP
DMOV      D003166 D002004	// L_4th BD Z ¢¬nC¡Í¨ùO¥ì¥ì
; L44
LOAD NOT  M00600	// EMERGENCY ALARM
AND NOT   D001000.6	// L_4th BD Z SVD BUSY
AND NOT   D001000.A	// L_4th BD Z WARNING
AND NOT   D001000.B	// L_4th BD Z MODULE ERR
AND NOT   D001000.C	// L_4th BD Z SVD ERR
AND NOT   M02011	// T)L_4th_ 01 Z JOG-
AND NOT   M02012	// T)L_4th_ 01 Z JOG+
AND NOT   M02013	// T)L_4th_ 01 Z SERVO ON
AND NOT   M0301C	// L_4th_01 Z Pos HOME >
AND NOT   M00613	// L_4th_01 BD Z NOT MV
NOT
OUT       M0151C	// L_4th BD Z HOLD CUT

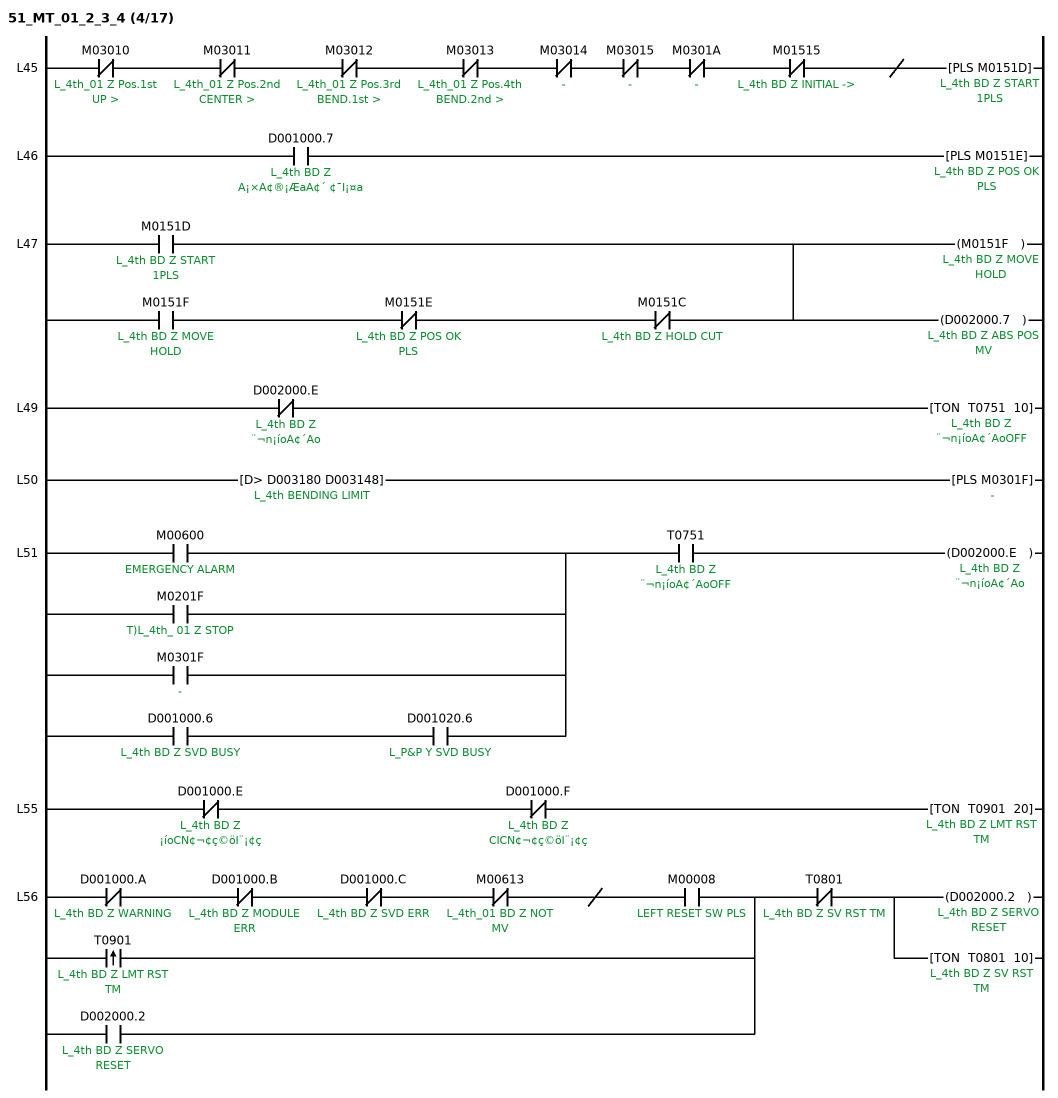
; L45
LOAD NOT  M03010	// L_4th_01 Z Pos.1st     UP >
AND NOT   M03011	// L_4th_01 Z Pos.2nd CENTER >
AND NOT   M03012	// L_4th_01 Z Pos.3rd BEND.1st >
AND NOT   M03013	// L_4th_01 Z Pos.4th BEND.2nd >
AND NOT   M03014	// -
AND NOT   M03015	// -
AND NOT   M0301A	// -
AND NOT   M01515	// L_4th BD Z INITIAL ->
NOT
OUTP      M0151D	// L_4th BD Z START 1PLS
; L46
LOAD      D001000.7	// L_4th BD Z A¡×A¢®¡ÆaA¢´ ¢¯I¡¤a
OUTP      M0151E	// L_4th BD Z POS OK PLS
; L47
LOAD      M0151D	// L_4th BD Z START 1PLS
LOAD      M0151F	// L_4th BD Z MOVE HOLD
AND NOT   M0151E	// L_4th BD Z POS OK PLS
AND NOT   M0151C	// L_4th BD Z HOLD CUT
OR LOAD
OUT       M0151F	// L_4th BD Z MOVE HOLD
OUT       D002000.7	// L_4th BD Z ABS POS MV
; L49
LOAD NOT  D002000.E	// L_4th BD Z ¨¬n¡íoA¢´Ao
TON       T0751 10	// L_4th BD Z ¨¬n¡íoA¢´AoOFF
; L50
LOADD>    D003180 D003148	// L_4th BENDING LIMIT
OUTP      M0301F	// -
; L51
LOAD      M00600	// EMERGENCY ALARM
OR        M0201F	// T)L_4th_ 01 Z STOP
OR        M0301F	// -
LOAD      D001000.6	// L_4th BD Z SVD BUSY
AND       D001020.6	// L_P&P Y SVD BUSY
OR LOAD
AND       T0751	// L_4th BD Z ¨¬n¡íoA¢´AoOFF
OUT       D002000.E	// L_4th BD Z ¨¬n¡íoA¢´Ao
; L55
LOAD NOT  D001000.E	// L_4th BD Z ¡íoCN¢¬¢ç©öI¨¡¢ç
AND NOT   D001000.F	// L_4th BD Z CICN¢¬¢ç©öI¨¡¢ç
TON       T0901 20	// L_4th BD Z LMT RST TM
; L56
LOAD NOT  D001000.A	// L_4th BD Z WARNING
AND NOT   D001000.B	// L_4th BD Z MODULE ERR
AND NOT   D001000.C	// L_4th BD Z SVD ERR
AND NOT   M00613	// L_4th_01 BD Z NOT MV
NOT
AND       M00008	// LEFT RESET SW PLS
ORP       T0901	// L_4th BD Z LMT RST TM
OR        D002000.2	// L_4th BD Z SERVO RESET
AND NOT   T0801	// L_4th BD Z SV RST TM
OUT       D002000.2	// L_4th BD Z SERVO RESET
TON       T0801 10	// L_4th BD Z SV RST TM

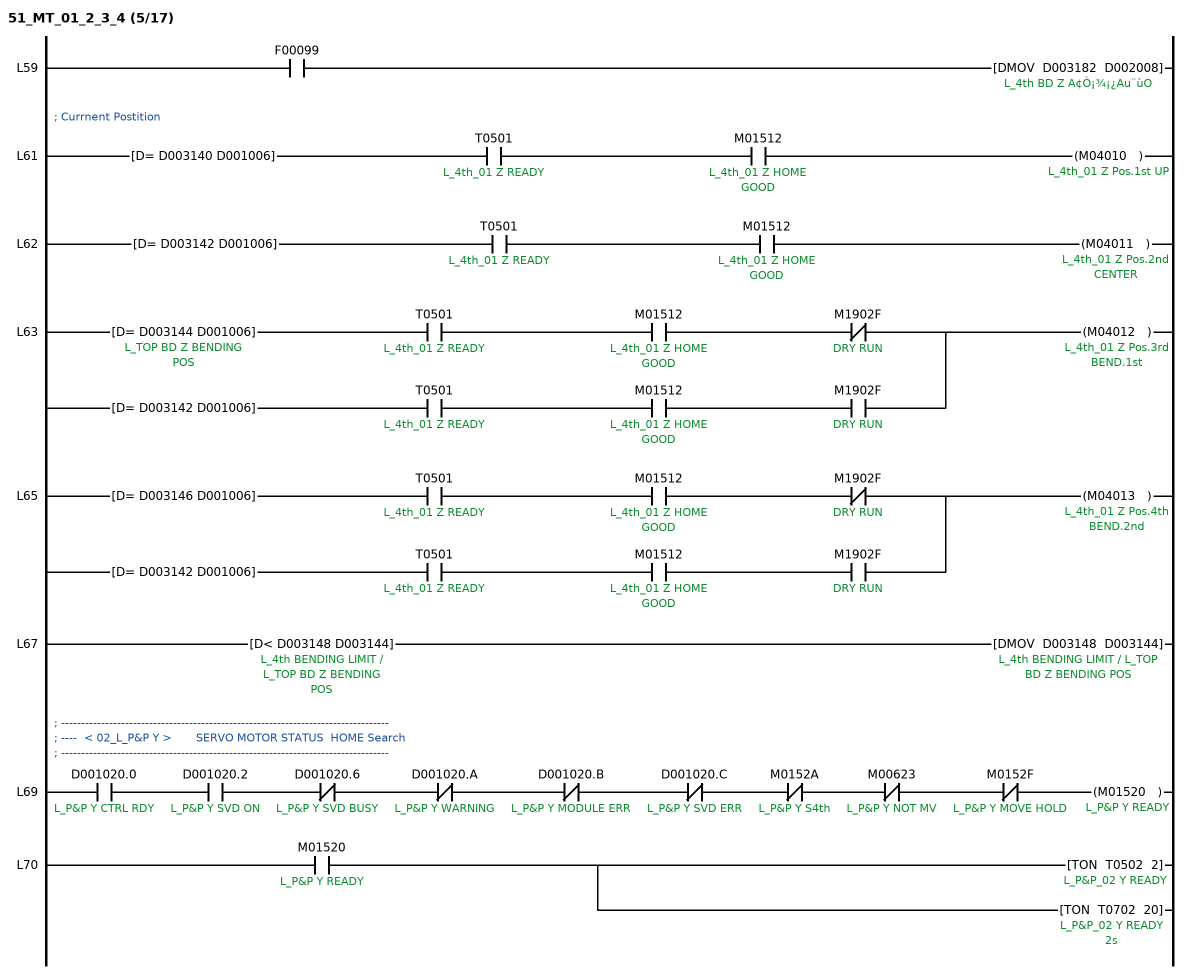
; L59
LOAD      F00099
DMOV      D003182 D002008	// L_4th BD Z A¢Ò¡¾¡¿Au¨ùO
// Currnent Postition
; L61
LOADD=    D003140 D001006
AND       T0501	// L_4th_01 Z READY
AND       M01512	// L_4th_01 Z HOME GOOD
OUT       M04010	// L_4th_01 Z Pos.1st UP
; L62
LOADD=    D003142 D001006
AND       T0501	// L_4th_01 Z READY
AND       M01512	// L_4th_01 Z HOME GOOD
OUT       M04011	// L_4th_01 Z Pos.2nd CENTER
; L63
LOADD=    D003144 D001006	// L_TOP BD Z BENDING POS
AND       T0501	// L_4th_01 Z READY
AND       M01512	// L_4th_01 Z HOME GOOD
AND NOT   M1902F	// DRY RUN
LOADD=    D003142 D001006
AND       T0501	// L_4th_01 Z READY
AND       M01512	// L_4th_01 Z HOME GOOD
AND       M1902F	// DRY RUN
OR LOAD
OUT       M04012	// L_4th_01 Z Pos.3rd BEND.1st
; L65
LOADD=    D003146 D001006
AND       T0501	// L_4th_01 Z READY
AND       M01512	// L_4th_01 Z HOME GOOD
AND NOT   M1902F	// DRY RUN
LOADD=    D003142 D001006
AND       T0501	// L_4th_01 Z READY
AND       M01512	// L_4th_01 Z HOME GOOD
AND       M1902F	// DRY RUN
OR LOAD
OUT       M04013	// L_4th_01 Z Pos.4th BEND.2nd
; L67
LOADD<    D003148 D003144	// L_4th BENDING LIMIT / L_TOP BD Z BENDING POS
DMOV      D003148 D003144	// L_4th BENDING LIMIT / L_TOP BD Z BENDING POS
// ----------------------------------------------------------------------------------
// 
// ----  < 02_L_P&P Y >       SERVO MOTOR STATUS  HOME Search
// 
// ----------------------------------------------------------------------------------
; L69
LOAD      D001020.0	// L_P&P Y CTRL RDY
AND       D001020.2	// L_P&P Y SVD ON
AND NOT   D001020.6	// L_P&P Y SVD BUSY
AND NOT   D001020.A	// L_P&P Y WARNING
AND NOT   D001020.B	// L_P&P Y MODULE ERR
AND NOT   D001020.C	// L_P&P Y SVD ERR
AND NOT   M0152A	// L_P&P Y S4th
AND NOT   M00623	// L_P&P Y NOT MV
AND NOT   M0152F	// L_P&P Y MOVE HOLD
OUT       M01520	// L_P&P Y READY
; L70
LOAD      M01520	// L_P&P Y READY
TON       T0502 2	// L_P&P_02 Y READY
TON       T0702 20	// L_P&P_02 Y READY 2s

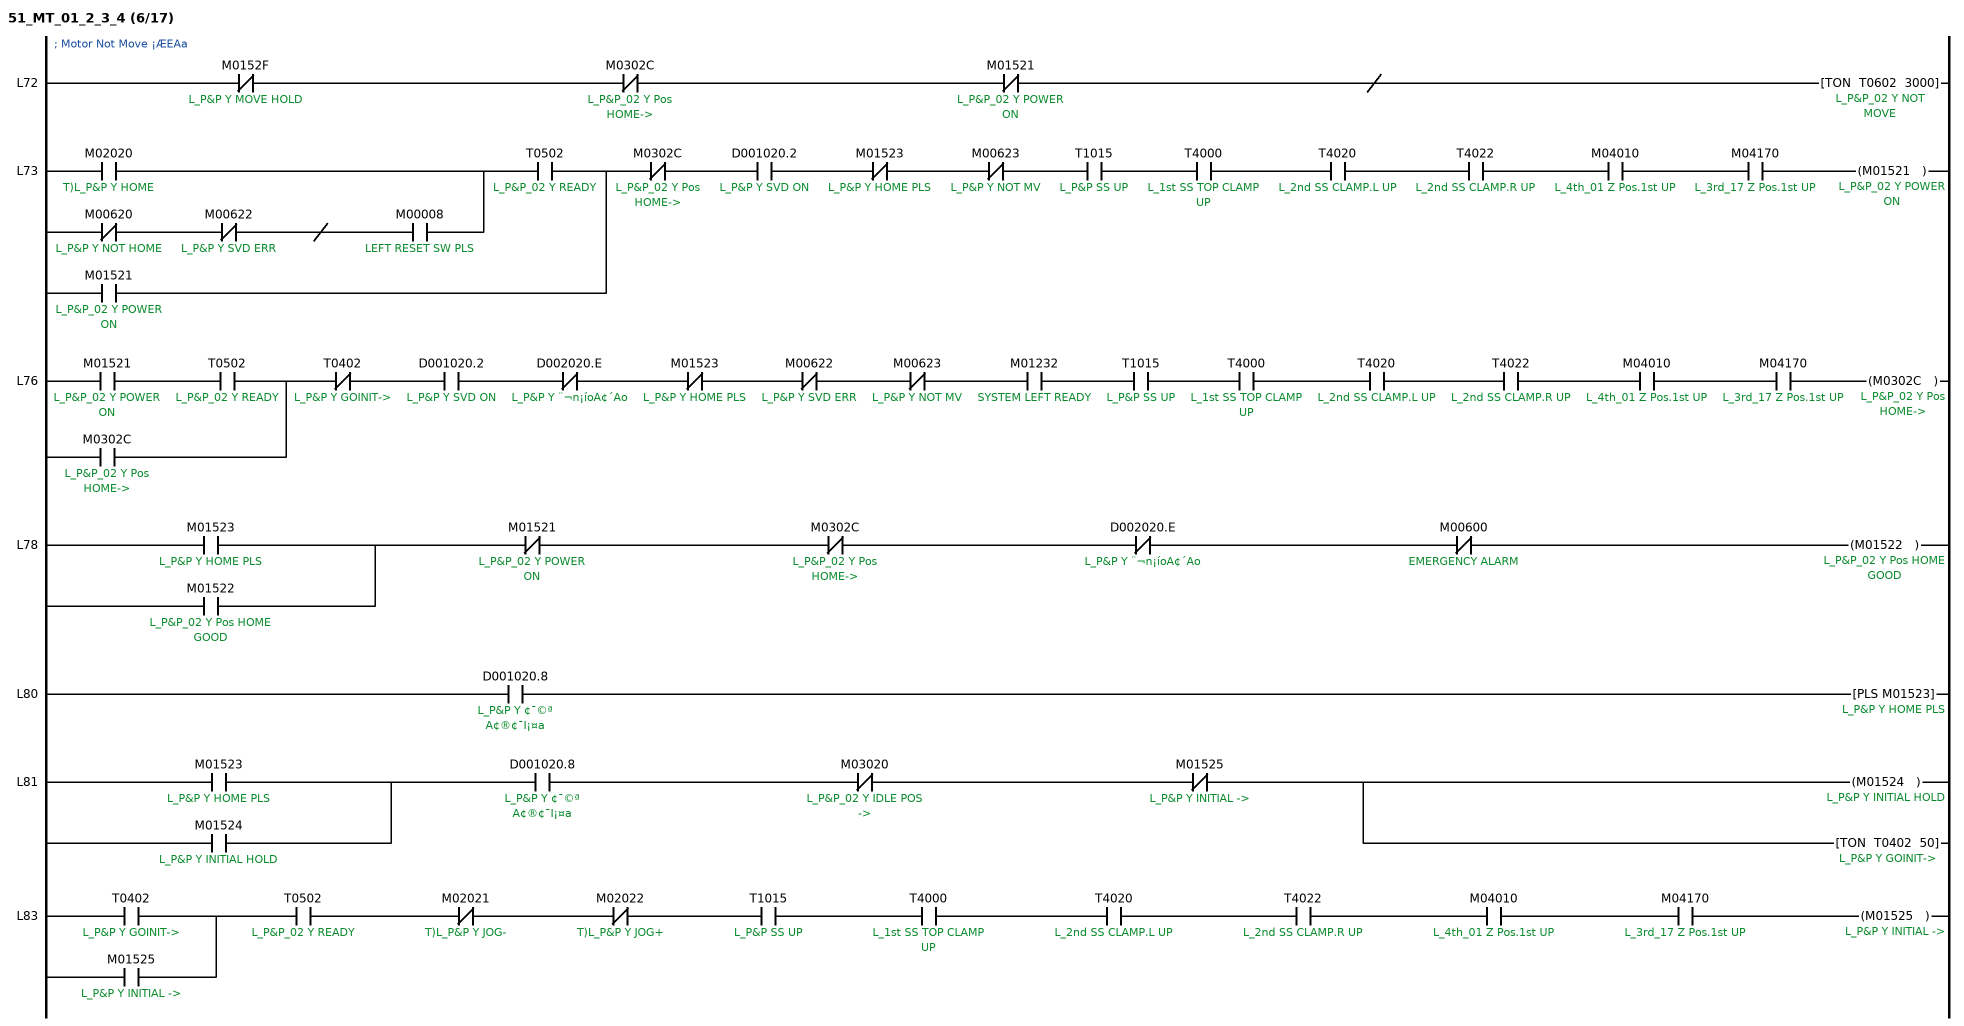
; L72
LOAD NOT  M0152F	// L_P&P Y MOVE HOLD
AND NOT   M0302C	// L_P&P_02 Y Pos HOME->
AND NOT   M01521	// L_P&P_02 Y POWER ON
NOT
TON       T0602 3000	// L_P&P_02 Y NOT MOVE
// output comment: Motor Not Move ¡ÆEAa
; L73
LOAD      M02020	// T)L_P&P Y HOME
LOAD NOT  M00620	// L_P&P Y NOT HOME
AND NOT   M00622	// L_P&P Y SVD ERR
NOT
AND       M00008	// LEFT RESET SW PLS
OR LOAD
AND       T0502	// L_P&P_02 Y READY
OR        M01521	// L_P&P_02 Y POWER ON
AND NOT   M0302C	// L_P&P_02 Y Pos HOME->
AND       D001020.2	// L_P&P Y SVD ON
AND NOT   M01523	// L_P&P Y HOME PLS
AND NOT   M00623	// L_P&P Y NOT MV
AND       T1015	// L_P&P SS UP
AND       T4000	// L_1st SS TOP CLAMP    UP
AND       T4020	// L_2nd SS CLAMP.L UP
AND       T4022	// L_2nd SS CLAMP.R UP
AND       M04010	// L_4th_01 Z Pos.1st UP
AND       M04170	// L_3rd_17 Z Pos.1st UP
OUT       M01521	// L_P&P_02 Y POWER ON
; L76
LOAD      M01521	// L_P&P_02 Y POWER ON
AND       T0502	// L_P&P_02 Y READY
OR        M0302C	// L_P&P_02 Y Pos HOME->
AND NOT   T0402	// L_P&P Y GOINIT->
AND       D001020.2	// L_P&P Y SVD ON
AND NOT   D002020.E	// L_P&P Y ¨¬n¡íoA¢´Ao
AND NOT   M01523	// L_P&P Y HOME PLS
AND NOT   M00622	// L_P&P Y SVD ERR
AND NOT   M00623	// L_P&P Y NOT MV
AND       M01232	// SYSTEM LEFT READY
AND       T1015	// L_P&P SS UP
AND       T4000	// L_1st SS TOP CLAMP    UP
AND       T4020	// L_2nd SS CLAMP.L UP
AND       T4022	// L_2nd SS CLAMP.R UP
AND       M04010	// L_4th_01 Z Pos.1st UP
AND       M04170	// L_3rd_17 Z Pos.1st UP
OUT       M0302C	// L_P&P_02 Y Pos HOME->
; L78
LOAD      M01523	// L_P&P Y HOME PLS
OR        M01522	// L_P&P_02 Y Pos HOME GOOD
AND NOT   M01521	// L_P&P_02 Y POWER ON
AND NOT   M0302C	// L_P&P_02 Y Pos HOME->
AND NOT   D002020.E	// L_P&P Y ¨¬n¡íoA¢´Ao
AND NOT   M00600	// EMERGENCY ALARM
OUT       M01522	// L_P&P_02 Y Pos HOME GOOD
; L80
LOAD      D001020.8	// L_P&P Y ¢¯©ªA¢®¢¯I¡¤a
OUTP      M01523	// L_P&P Y HOME PLS
; L81
LOAD      M01523	// L_P&P Y HOME PLS
OR        M01524	// L_P&P Y INITIAL HOLD
AND       D001020.8	// L_P&P Y ¢¯©ªA¢®¢¯I¡¤a
AND NOT   M03020	// L_P&P_02 Y IDLE POS ->
AND NOT   M01525	// L_P&P Y INITIAL ->
OUT       M01524	// L_P&P Y INITIAL HOLD
TON       T0402 50	// L_P&P Y GOINIT->
; L83
LOAD      T0402	// L_P&P Y GOINIT->
OR        M01525	// L_P&P Y INITIAL ->
AND       T0502	// L_P&P_02 Y READY
AND NOT   M02021	// T)L_P&P Y JOG-
AND NOT   M02022	// T)L_P&P Y JOG+
AND       T1015	// L_P&P SS UP
AND       T4000	// L_1st SS TOP CLAMP    UP
AND       T4020	// L_2nd SS CLAMP.L UP
AND       T4022	// L_2nd SS CLAMP.R UP
AND       M04010	// L_4th_01 Z Pos.1st UP
AND       M04170	// L_3rd_17 Z Pos.1st UP
OUT       M01525	// L_P&P Y INITIAL ->

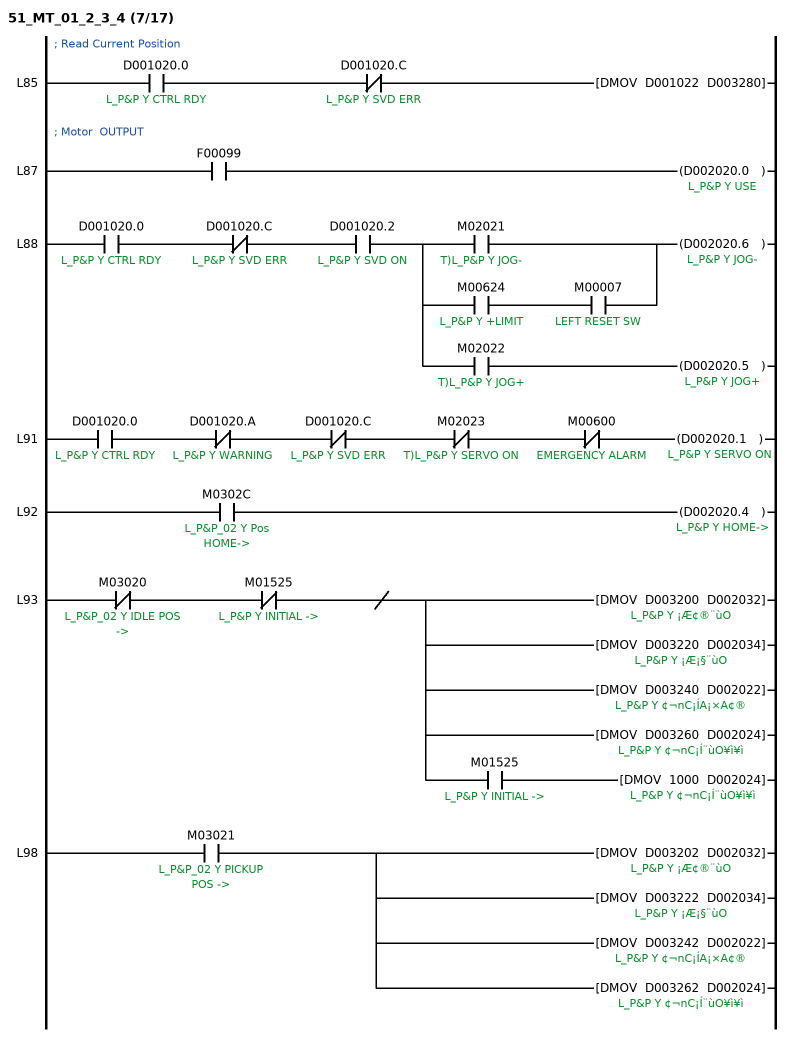
; L85
LOAD      D001020.0	// L_P&P Y CTRL RDY
AND NOT   D001020.C	// L_P&P Y SVD ERR
DMOV      D001022 D003280
// output comment: Read Current Position
//  Motor  OUTPUT
; L87
LOAD      F00099
OUT       D002020.0	// L_P&P Y USE
; L88
LOAD      D001020.0	// L_P&P Y CTRL RDY
AND NOT   D001020.C	// L_P&P Y SVD ERR
AND       D001020.2	// L_P&P Y SVD ON
MPUSH
LOAD      M02021	// T)L_P&P Y JOG-
LOAD      M00624	// L_P&P Y +LIMIT
AND       M00007	// LEFT RESET SW
OR LOAD
AND LOAD
OUT       D002020.6	// L_P&P Y JOG-
MPOP
AND       M02022	// T)L_P&P Y JOG+
OUT       D002020.5	// L_P&P Y JOG+
; L91
LOAD      D001020.0	// L_P&P Y CTRL RDY
AND NOT   D001020.A	// L_P&P Y WARNING
AND NOT   D001020.C	// L_P&P Y SVD ERR
AND NOT   M02023	// T)L_P&P Y SERVO ON
AND NOT   M00600	// EMERGENCY ALARM
OUT       D002020.1	// L_P&P Y SERVO ON
; L92
LOAD      M0302C	// L_P&P_02 Y Pos HOME->
OUT       D002020.4	// L_P&P Y HOME->
; L93
LOAD NOT  M03020	// L_P&P_02 Y IDLE POS ->
AND NOT   M01525	// L_P&P Y INITIAL ->
NOT
DMOV      D003200 D002032	// L_P&P Y ¡Æ¢®¨ùO
DMOV      D003220 D002034	// L_P&P Y ¡Æ¡§¨ùO
DMOV      D003240 D002022	// L_P&P Y ¢¬nC¡ÍA¡×A¢®
DMOV      D003260 D002024	// L_P&P Y ¢¬nC¡Í¨ùO¥ì¥ì
AND       M01525	// L_P&P Y INITIAL ->
DMOV      1000 D002024	// L_P&P Y ¢¬nC¡Í¨ùO¥ì¥ì
; L98
LOAD      M03021	// L_P&P_02 Y PICKUP POS ->
DMOV      D003202 D002032	// L_P&P Y ¡Æ¢®¨ùO
DMOV      D003222 D002034	// L_P&P Y ¡Æ¡§¨ùO
DMOV      D003242 D002022	// L_P&P Y ¢¬nC¡ÍA¡×A¢®
DMOV      D003262 D002024	// L_P&P Y ¢¬nC¡Í¨ùO¥ì¥ì

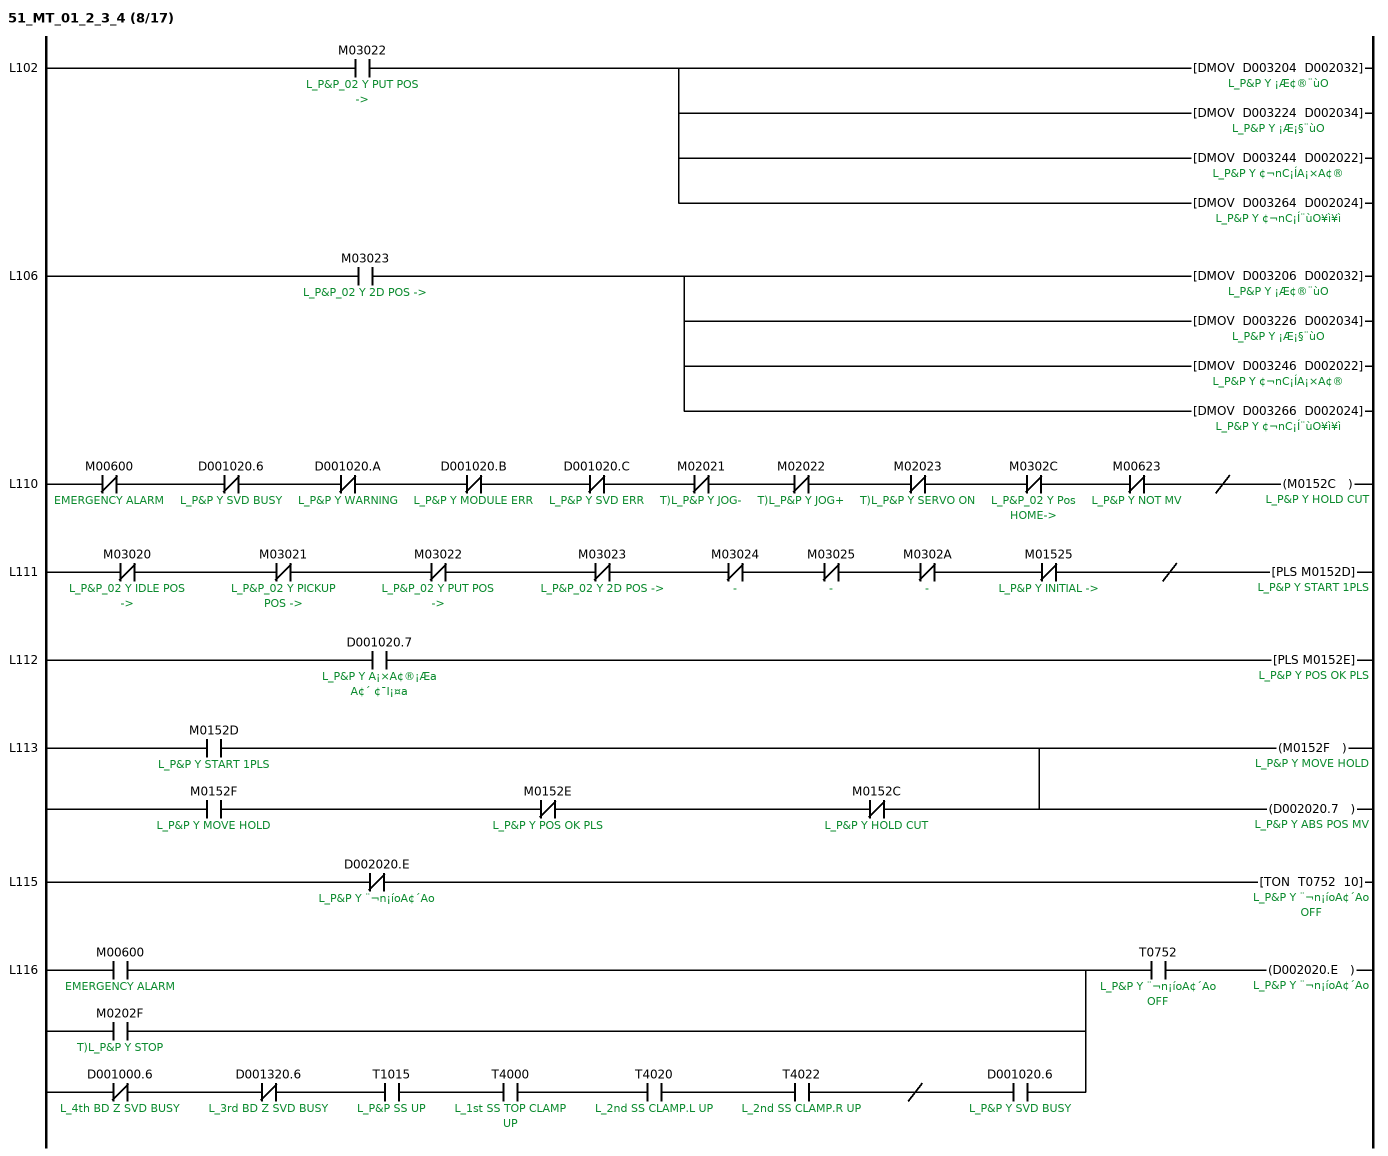
; L102
LOAD      M03022	// L_P&P_02 Y PUT POS ->
DMOV      D003204 D002032	// L_P&P Y ¡Æ¢®¨ùO
DMOV      D003224 D002034	// L_P&P Y ¡Æ¡§¨ùO
DMOV      D003244 D002022	// L_P&P Y ¢¬nC¡ÍA¡×A¢®
DMOV      D003264 D002024	// L_P&P Y ¢¬nC¡Í¨ùO¥ì¥ì
; L106
LOAD      M03023	// L_P&P_02 Y 2D POS ->
DMOV      D003206 D002032	// L_P&P Y ¡Æ¢®¨ùO
DMOV      D003226 D002034	// L_P&P Y ¡Æ¡§¨ùO
DMOV      D003246 D002022	// L_P&P Y ¢¬nC¡ÍA¡×A¢®
DMOV      D003266 D002024	// L_P&P Y ¢¬nC¡Í¨ùO¥ì¥ì
; L110
LOAD NOT  M00600	// EMERGENCY ALARM
AND NOT   D001020.6	// L_P&P Y SVD BUSY
AND NOT   D001020.A	// L_P&P Y WARNING
AND NOT   D001020.B	// L_P&P Y MODULE ERR
AND NOT   D001020.C	// L_P&P Y SVD ERR
AND NOT   M02021	// T)L_P&P Y JOG-
AND NOT   M02022	// T)L_P&P Y JOG+
AND NOT   M02023	// T)L_P&P Y SERVO ON
AND NOT   M0302C	// L_P&P_02 Y Pos HOME->
AND NOT   M00623	// L_P&P Y NOT MV
NOT
OUT       M0152C	// L_P&P Y HOLD CUT
; L111
LOAD NOT  M03020	// L_P&P_02 Y IDLE POS ->
AND NOT   M03021	// L_P&P_02 Y PICKUP POS ->
AND NOT   M03022	// L_P&P_02 Y PUT POS ->
AND NOT   M03023	// L_P&P_02 Y 2D POS ->
AND NOT   M03024	// -
AND NOT   M03025	// -
AND NOT   M0302A	// -
AND NOT   M01525	// L_P&P Y INITIAL ->
NOT
OUTP      M0152D	// L_P&P Y START 1PLS
; L112
LOAD      D001020.7	// L_P&P Y A¡×A¢®¡ÆaA¢´ ¢¯I¡¤a
OUTP      M0152E	// L_P&P Y POS OK PLS
; L113
LOAD      M0152D	// L_P&P Y START 1PLS
LOAD      M0152F	// L_P&P Y MOVE HOLD
AND NOT   M0152E	// L_P&P Y POS OK PLS
AND NOT   M0152C	// L_P&P Y HOLD CUT
OR LOAD
OUT       M0152F	// L_P&P Y MOVE HOLD
OUT       D002020.7	// L_P&P Y ABS POS MV
; L115
LOAD NOT  D002020.E	// L_P&P Y ¨¬n¡íoA¢´Ao
TON       T0752 10	// L_P&P Y ¨¬n¡íoA¢´AoOFF
; L116
LOAD      M00600	// EMERGENCY ALARM
OR        M0202F	// T)L_P&P Y STOP
LOAD NOT  D001000.6	// L_4th BD Z SVD BUSY
AND NOT   D001320.6	// L_3rd BD Z SVD BUSY
AND       T1015	// L_P&P SS UP
AND       T4000	// L_1st SS TOP CLAMP    UP
AND       T4020	// L_2nd SS CLAMP.L UP
AND       T4022	// L_2nd SS CLAMP.R UP
NOT
AND       D001020.6	// L_P&P Y SVD BUSY
OR LOAD
AND       T0752	// L_P&P Y ¨¬n¡íoA¢´AoOFF
OUT       D002020.E	// L_P&P Y ¨¬n¡íoA¢´Ao

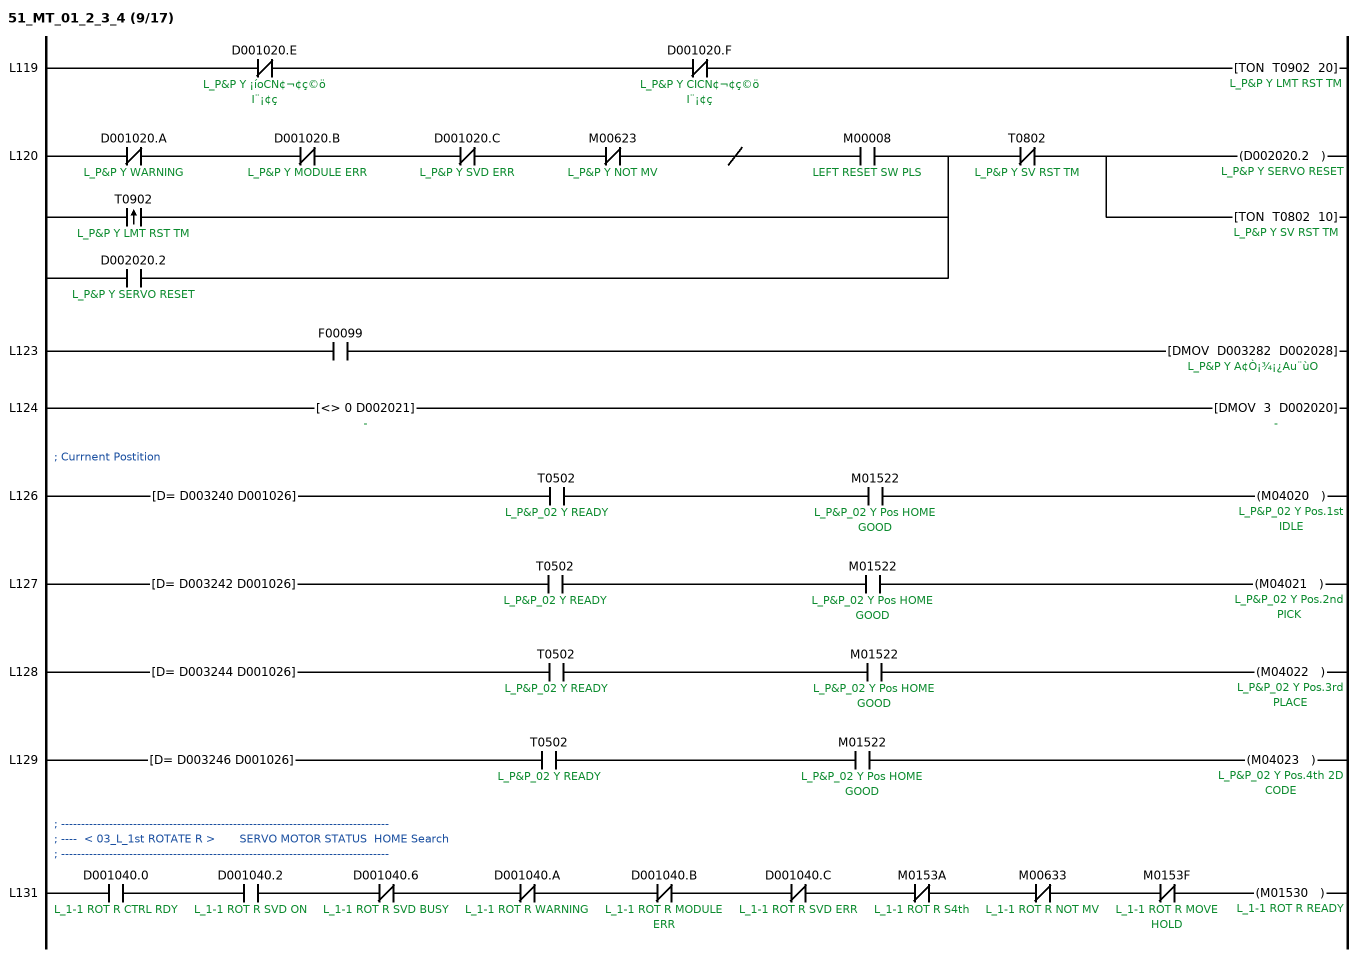
; L119
LOAD NOT  D001020.E	// L_P&P Y ¡íoCN¢¬¢ç©öI¨¡¢ç
AND NOT   D001020.F	// L_P&P Y CICN¢¬¢ç©öI¨¡¢ç
TON       T0902 20	// L_P&P Y LMT RST TM
; L120
LOAD NOT  D001020.A	// L_P&P Y WARNING
AND NOT   D001020.B	// L_P&P Y MODULE ERR
AND NOT   D001020.C	// L_P&P Y SVD ERR
AND NOT   M00623	// L_P&P Y NOT MV
NOT
AND       M00008	// LEFT RESET SW PLS
ORP       T0902	// L_P&P Y LMT RST TM
OR        D002020.2	// L_P&P Y SERVO RESET
AND NOT   T0802	// L_P&P Y SV RST TM
OUT       D002020.2	// L_P&P Y SERVO RESET
TON       T0802 10	// L_P&P Y SV RST TM
; L123
LOAD      F00099
DMOV      D003282 D002028	// L_P&P Y A¢Ò¡¾¡¿Au¨ùO
; L124
LOAD<>    0 D002021	// -
DMOV      3 D002020	// -
// Currnent Postition
; L126
LOADD=    D003240 D001026
AND       T0502	// L_P&P_02 Y READY
AND       M01522	// L_P&P_02 Y Pos HOME GOOD
OUT       M04020	// L_P&P_02 Y Pos.1st IDLE
; L127
LOADD=    D003242 D001026
AND       T0502	// L_P&P_02 Y READY
AND       M01522	// L_P&P_02 Y Pos HOME GOOD
OUT       M04021	// L_P&P_02 Y Pos.2nd PICK
; L128
LOADD=    D003244 D001026
AND       T0502	// L_P&P_02 Y READY
AND       M01522	// L_P&P_02 Y Pos HOME GOOD
OUT       M04022	// L_P&P_02 Y Pos.3rd PLACE
; L129
LOADD=    D003246 D001026
AND       T0502	// L_P&P_02 Y READY
AND       M01522	// L_P&P_02 Y Pos HOME GOOD
OUT       M04023	// L_P&P_02 Y Pos.4th 2D CODE
// ----------------------------------------------------------------------------------
// 
// ----  < 03_L_1st ROTATE R >       SERVO MOTOR STATUS  HOME Search
// 
// ----------------------------------------------------------------------------------
; L131
LOAD      D001040.0	// L_1-1 ROT R CTRL RDY
AND       D001040.2	// L_1-1 ROT R SVD ON
AND NOT   D001040.6	// L_1-1 ROT R SVD BUSY
AND NOT   D001040.A	// L_1-1 ROT R WARNING
AND NOT   D001040.B	// L_1-1 ROT R MODULE ERR
AND NOT   D001040.C	// L_1-1 ROT R SVD ERR
AND NOT   M0153A	// L_1-1 ROT R S4th
AND NOT   M00633	// L_1-1 ROT R NOT MV
AND NOT   M0153F	// L_1-1 ROT R MOVE HOLD
OUT       M01530	// L_1-1 ROT R READY

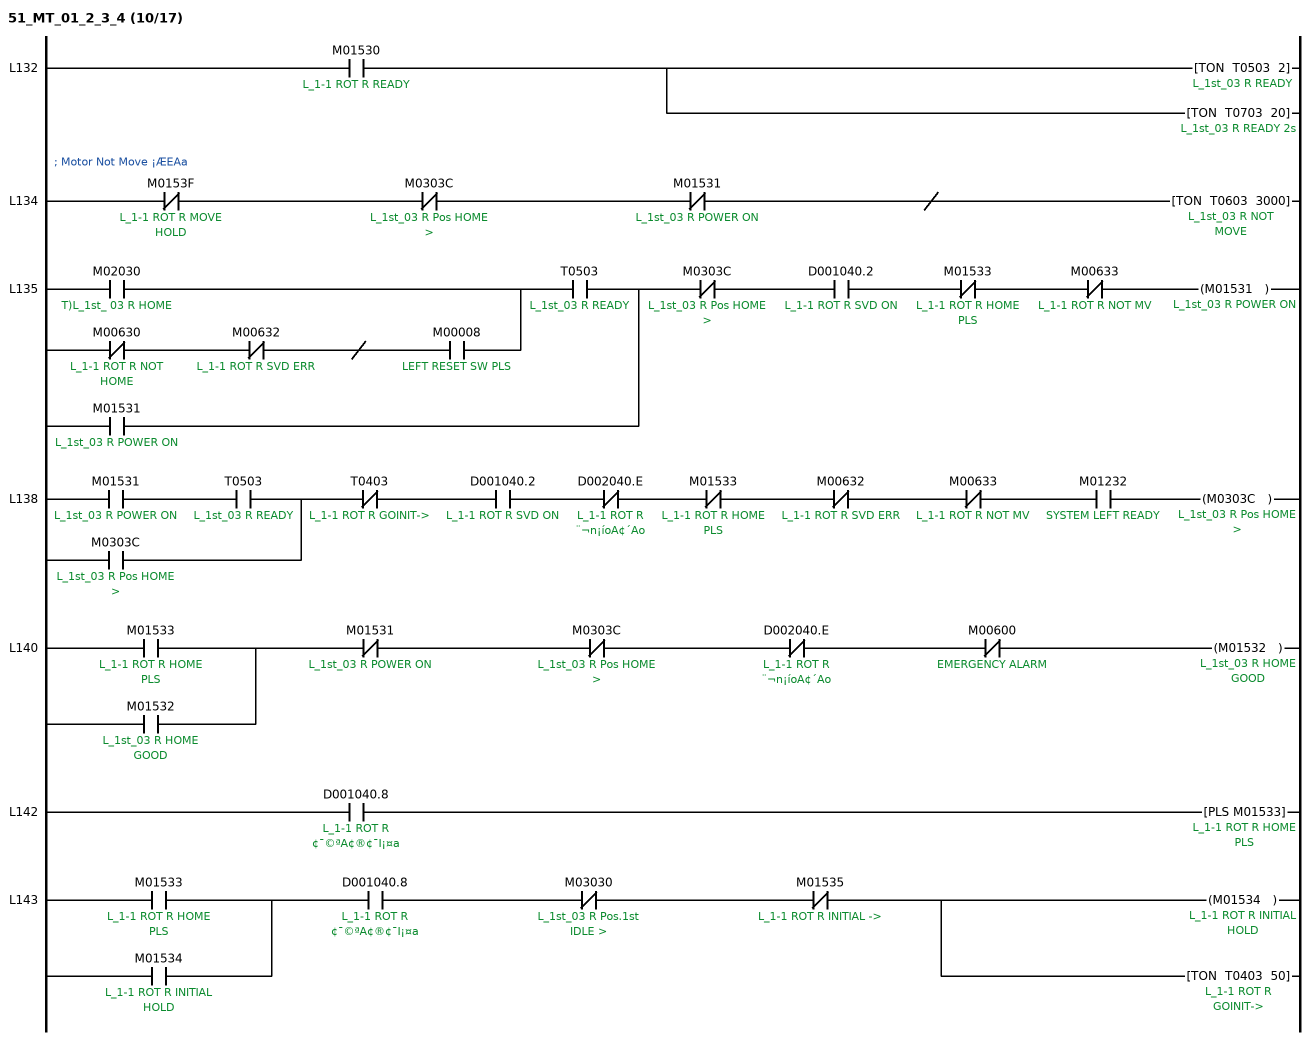
; L132
LOAD      M01530	// L_1-1 ROT R READY
TON       T0503 2	// L_1st_03 R READY
TON       T0703 20	// L_1st_03 R READY 2s
; L134
LOAD NOT  M0153F	// L_1-1 ROT R MOVE HOLD
AND NOT   M0303C	// L_1st_03 R Pos HOME >
AND NOT   M01531	// L_1st_03 R POWER ON
NOT
TON       T0603 3000	// L_1st_03 R NOT MOVE
// output comment: Motor Not Move ¡ÆEAa
; L135
LOAD      M02030	// T)L_1st_ 03 R HOME
LOAD NOT  M00630	// L_1-1 ROT R NOT HOME
AND NOT   M00632	// L_1-1 ROT R SVD ERR
NOT
AND       M00008	// LEFT RESET SW PLS
OR LOAD
AND       T0503	// L_1st_03 R READY
OR        M01531	// L_1st_03 R POWER ON
AND NOT   M0303C	// L_1st_03 R Pos HOME >
AND       D001040.2	// L_1-1 ROT R SVD ON
AND NOT   M01533	// L_1-1 ROT R HOME PLS
AND NOT   M00633	// L_1-1 ROT R NOT MV
OUT       M01531	// L_1st_03 R POWER ON
; L138
LOAD      M01531	// L_1st_03 R POWER ON
AND       T0503	// L_1st_03 R READY
OR        M0303C	// L_1st_03 R Pos HOME >
AND NOT   T0403	// L_1-1 ROT R GOINIT->
AND       D001040.2	// L_1-1 ROT R SVD ON
AND NOT   D002040.E	// L_1-1 ROT R ¨¬n¡íoA¢´Ao
AND NOT   M01533	// L_1-1 ROT R HOME PLS
AND NOT   M00632	// L_1-1 ROT R SVD ERR
AND NOT   M00633	// L_1-1 ROT R NOT MV
AND       M01232	// SYSTEM LEFT READY
OUT       M0303C	// L_1st_03 R Pos HOME >
; L140
LOAD      M01533	// L_1-1 ROT R HOME PLS
OR        M01532	// L_1st_03 R HOME GOOD
AND NOT   M01531	// L_1st_03 R POWER ON
AND NOT   M0303C	// L_1st_03 R Pos HOME >
AND NOT   D002040.E	// L_1-1 ROT R ¨¬n¡íoA¢´Ao
AND NOT   M00600	// EMERGENCY ALARM
OUT       M01532	// L_1st_03 R HOME GOOD
; L142
LOAD      D001040.8	// L_1-1 ROT R ¢¯©ªA¢®¢¯I¡¤a
OUTP      M01533	// L_1-1 ROT R HOME PLS
; L143
LOAD      M01533	// L_1-1 ROT R HOME PLS
OR        M01534	// L_1-1 ROT R INITIAL HOLD
AND       D001040.8	// L_1-1 ROT R ¢¯©ªA¢®¢¯I¡¤a
AND NOT   M03030	// L_1st_03 R Pos.1st IDLE >
AND NOT   M01535	// L_1-1 ROT R INITIAL ->
OUT       M01534	// L_1-1 ROT R INITIAL HOLD
TON       T0403 50	// L_1-1 ROT R GOINIT->

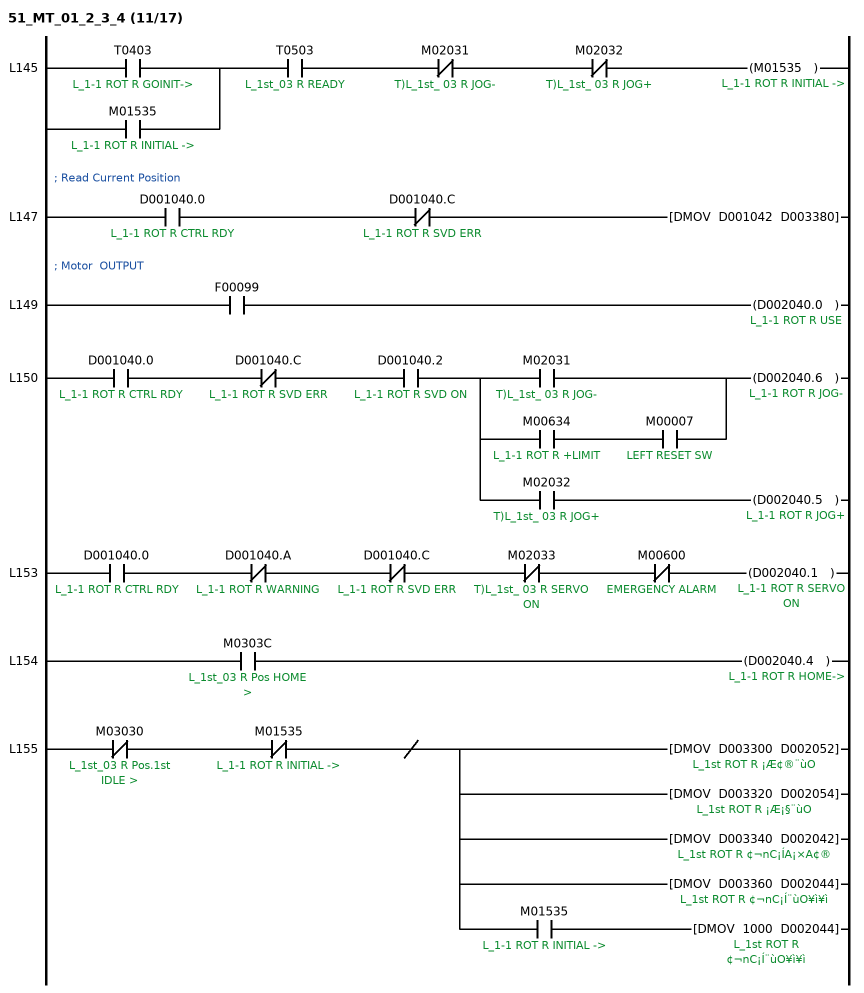
; L145
LOAD      T0403	// L_1-1 ROT R GOINIT->
OR        M01535	// L_1-1 ROT R INITIAL ->
AND       T0503	// L_1st_03 R READY
AND NOT   M02031	// T)L_1st_ 03 R JOG-
AND NOT   M02032	// T)L_1st_ 03 R JOG+
OUT       M01535	// L_1-1 ROT R INITIAL ->
; L147
LOAD      D001040.0	// L_1-1 ROT R CTRL RDY
AND NOT   D001040.C	// L_1-1 ROT R SVD ERR
DMOV      D001042 D003380
// output comment: Read Current Position
//  Motor  OUTPUT
; L149
LOAD      F00099
OUT       D002040.0	// L_1-1 ROT R USE
; L150
LOAD      D001040.0	// L_1-1 ROT R CTRL RDY
AND NOT   D001040.C	// L_1-1 ROT R SVD ERR
AND       D001040.2	// L_1-1 ROT R SVD ON
MPUSH
LOAD      M02031	// T)L_1st_ 03 R JOG-
LOAD      M00634	// L_1-1 ROT R +LIMIT
AND       M00007	// LEFT RESET SW
OR LOAD
AND LOAD
OUT       D002040.6	// L_1-1 ROT R JOG-
MPOP
AND       M02032	// T)L_1st_ 03 R JOG+
OUT       D002040.5	// L_1-1 ROT R JOG+
; L153
LOAD      D001040.0	// L_1-1 ROT R CTRL RDY
AND NOT   D001040.A	// L_1-1 ROT R WARNING
AND NOT   D001040.C	// L_1-1 ROT R SVD ERR
AND NOT   M02033	// T)L_1st_ 03 R SERVO ON
AND NOT   M00600	// EMERGENCY ALARM
OUT       D002040.1	// L_1-1 ROT R SERVO ON
; L154
LOAD      M0303C	// L_1st_03 R Pos HOME >
OUT       D002040.4	// L_1-1 ROT R HOME->
; L155
LOAD NOT  M03030	// L_1st_03 R Pos.1st IDLE >
AND NOT   M01535	// L_1-1 ROT R INITIAL ->
NOT
DMOV      D003300 D002052	// L_1st ROT R ¡Æ¢®¨ùO
DMOV      D003320 D002054	// L_1st ROT R ¡Æ¡§¨ùO
DMOV      D003340 D002042	// L_1st ROT R ¢¬nC¡ÍA¡×A¢®
DMOV      D003360 D002044	// L_1st ROT R ¢¬nC¡Í¨ùO¥ì¥ì
AND       M01535	// L_1-1 ROT R INITIAL ->
DMOV      1000 D002044	// L_1st ROT R ¢¬nC¡Í¨ùO¥ì¥ì

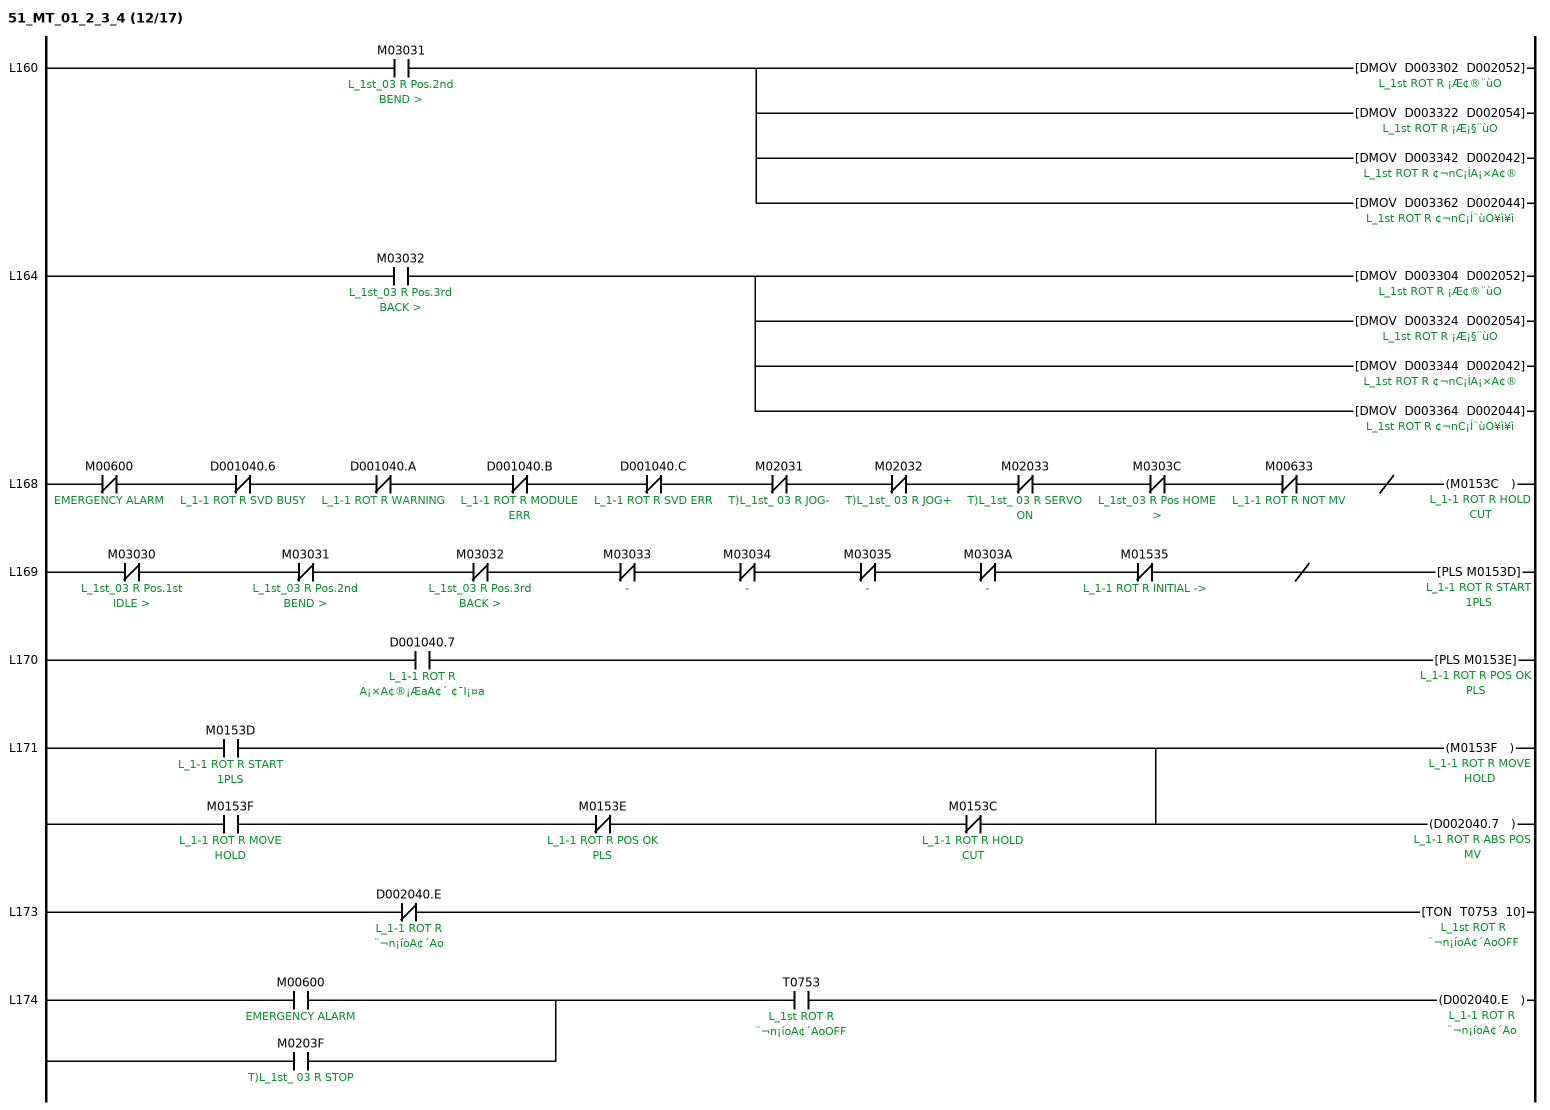
; L160
LOAD      M03031	// L_1st_03 R Pos.2nd BEND >
DMOV      D003302 D002052	// L_1st ROT R ¡Æ¢®¨ùO
DMOV      D003322 D002054	// L_1st ROT R ¡Æ¡§¨ùO
DMOV      D003342 D002042	// L_1st ROT R ¢¬nC¡ÍA¡×A¢®
DMOV      D003362 D002044	// L_1st ROT R ¢¬nC¡Í¨ùO¥ì¥ì
; L164
LOAD      M03032	// L_1st_03 R Pos.3rd BACK >
DMOV      D003304 D002052	// L_1st ROT R ¡Æ¢®¨ùO
DMOV      D003324 D002054	// L_1st ROT R ¡Æ¡§¨ùO
DMOV      D003344 D002042	// L_1st ROT R ¢¬nC¡ÍA¡×A¢®
DMOV      D003364 D002044	// L_1st ROT R ¢¬nC¡Í¨ùO¥ì¥ì
; L168
LOAD NOT  M00600	// EMERGENCY ALARM
AND NOT   D001040.6	// L_1-1 ROT R SVD BUSY
AND NOT   D001040.A	// L_1-1 ROT R WARNING
AND NOT   D001040.B	// L_1-1 ROT R MODULE ERR
AND NOT   D001040.C	// L_1-1 ROT R SVD ERR
AND NOT   M02031	// T)L_1st_ 03 R JOG-
AND NOT   M02032	// T)L_1st_ 03 R JOG+
AND NOT   M02033	// T)L_1st_ 03 R SERVO ON
AND NOT   M0303C	// L_1st_03 R Pos HOME >
AND NOT   M00633	// L_1-1 ROT R NOT MV
NOT
OUT       M0153C	// L_1-1 ROT R HOLD CUT
; L169
LOAD NOT  M03030	// L_1st_03 R Pos.1st IDLE >
AND NOT   M03031	// L_1st_03 R Pos.2nd BEND >
AND NOT   M03032	// L_1st_03 R Pos.3rd BACK >
AND NOT   M03033	// -
AND NOT   M03034	// -
AND NOT   M03035	// -
AND NOT   M0303A	// -
AND NOT   M01535	// L_1-1 ROT R INITIAL ->
NOT
OUTP      M0153D	// L_1-1 ROT R START 1PLS
; L170
LOAD      D001040.7	// L_1-1 ROT R A¡×A¢®¡ÆaA¢´ ¢¯I¡¤a
OUTP      M0153E	// L_1-1 ROT R POS OK PLS
; L171
LOAD      M0153D	// L_1-1 ROT R START 1PLS
LOAD      M0153F	// L_1-1 ROT R MOVE HOLD
AND NOT   M0153E	// L_1-1 ROT R POS OK PLS
AND NOT   M0153C	// L_1-1 ROT R HOLD CUT
OR LOAD
OUT       M0153F	// L_1-1 ROT R MOVE HOLD
OUT       D002040.7	// L_1-1 ROT R ABS POS MV
; L173
LOAD NOT  D002040.E	// L_1-1 ROT R ¨¬n¡íoA¢´Ao
TON       T0753 10	// L_1st ROT R ¨¬n¡íoA¢´AoOFF
; L174
LOAD      M00600	// EMERGENCY ALARM
OR        M0203F	// T)L_1st_ 03 R STOP
AND       T0753	// L_1st ROT R ¨¬n¡íoA¢´AoOFF
OUT       D002040.E	// L_1-1 ROT R ¨¬n¡íoA¢´Ao

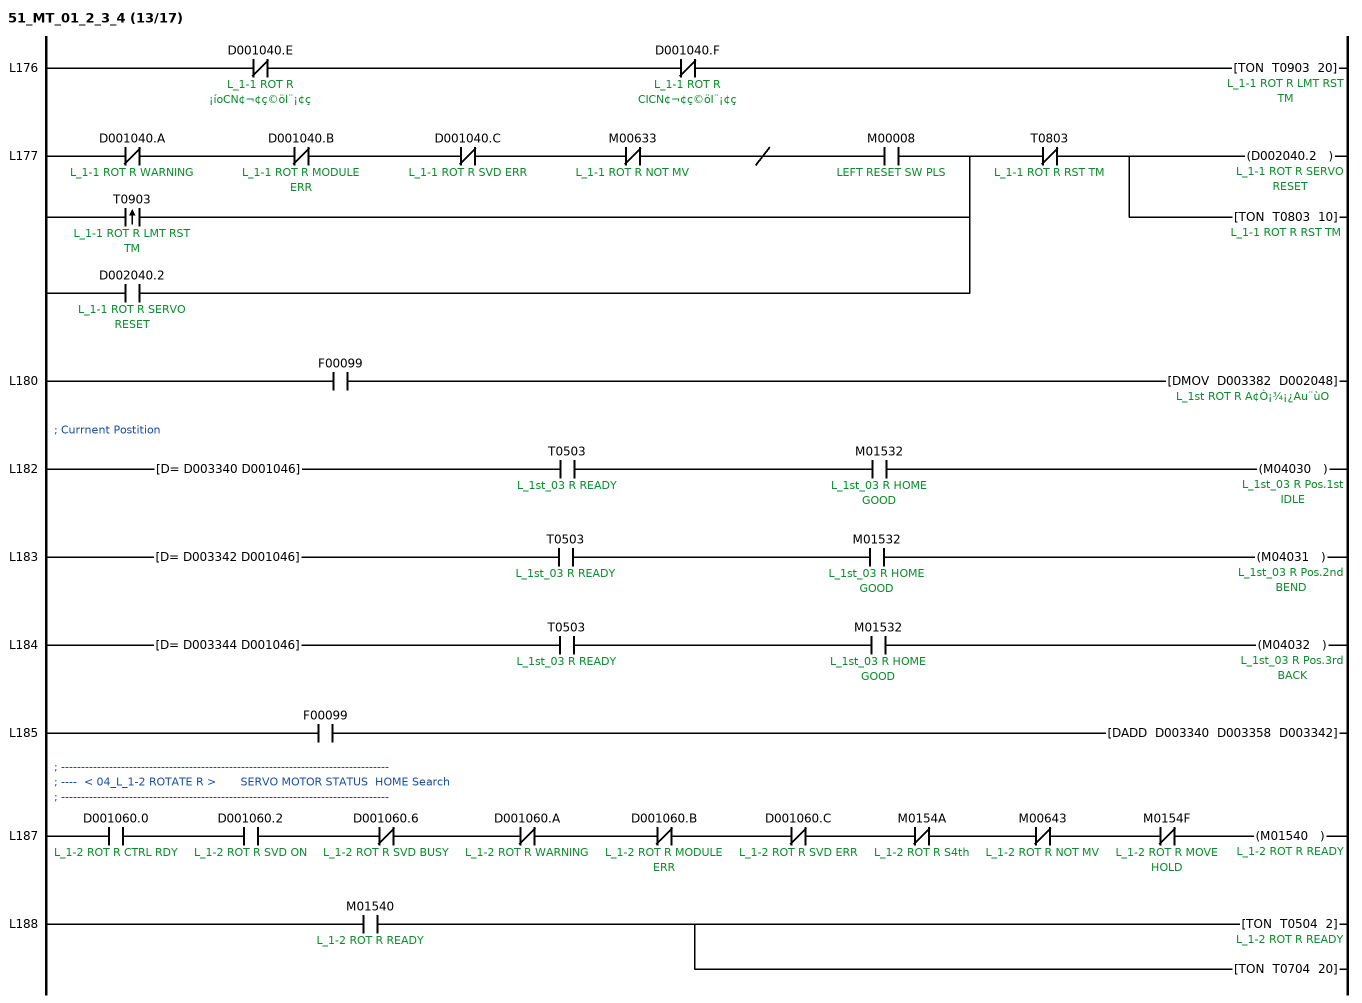
; L176
LOAD NOT  D001040.E	// L_1-1 ROT R ¡íoCN¢¬¢ç©öI¨¡¢ç
AND NOT   D001040.F	// L_1-1 ROT R CICN¢¬¢ç©öI¨¡¢ç
TON       T0903 20	// L_1-1 ROT R LMT RST TM
; L177
LOAD NOT  D001040.A	// L_1-1 ROT R WARNING
AND NOT   D001040.B	// L_1-1 ROT R MODULE ERR
AND NOT   D001040.C	// L_1-1 ROT R SVD ERR
AND NOT   M00633	// L_1-1 ROT R NOT MV
NOT
AND       M00008	// LEFT RESET SW PLS
ORP       T0903	// L_1-1 ROT R LMT RST TM
OR        D002040.2	// L_1-1 ROT R SERVO RESET
AND NOT   T0803	// L_1-1 ROT R RST TM
OUT       D002040.2	// L_1-1 ROT R SERVO RESET
TON       T0803 10	// L_1-1 ROT R RST TM
; L180
LOAD      F00099
DMOV      D003382 D002048	// L_1st ROT R A¢Ò¡¾¡¿Au¨ùO
// Currnent Postition
; L182
LOADD=    D003340 D001046
AND       T0503	// L_1st_03 R READY
AND       M01532	// L_1st_03 R HOME GOOD
OUT       M04030	// L_1st_03 R Pos.1st IDLE
; L183
LOADD=    D003342 D001046
AND       T0503	// L_1st_03 R READY
AND       M01532	// L_1st_03 R HOME GOOD
OUT       M04031	// L_1st_03 R Pos.2nd BEND
; L184
LOADD=    D003344 D001046
AND       T0503	// L_1st_03 R READY
AND       M01532	// L_1st_03 R HOME GOOD
OUT       M04032	// L_1st_03 R Pos.3rd BACK
; L185
LOAD      F00099
DADD      D003340 D003358 D003342
// ----------------------------------------------------------------------------------
// 
// ----  < 04_L_1-2 ROTATE R >       SERVO MOTOR STATUS  HOME Search
// 
// ----------------------------------------------------------------------------------
; L187
LOAD      D001060.0	// L_1-2 ROT R CTRL RDY
AND       D001060.2	// L_1-2 ROT R SVD ON
AND NOT   D001060.6	// L_1-2 ROT R SVD BUSY
AND NOT   D001060.A	// L_1-2 ROT R WARNING
AND NOT   D001060.B	// L_1-2 ROT R MODULE ERR
AND NOT   D001060.C	// L_1-2 ROT R SVD ERR
AND NOT   M0154A	// L_1-2 ROT R S4th
AND NOT   M00643	// L_1-2 ROT R NOT MV
AND NOT   M0154F	// L_1-2 ROT R MOVE HOLD
OUT       M01540	// L_1-2 ROT R READY
; L188
LOAD      M01540	// L_1-2 ROT R READY
TON       T0504 2	// L_1-2 ROT R READY
TON       T0704 20

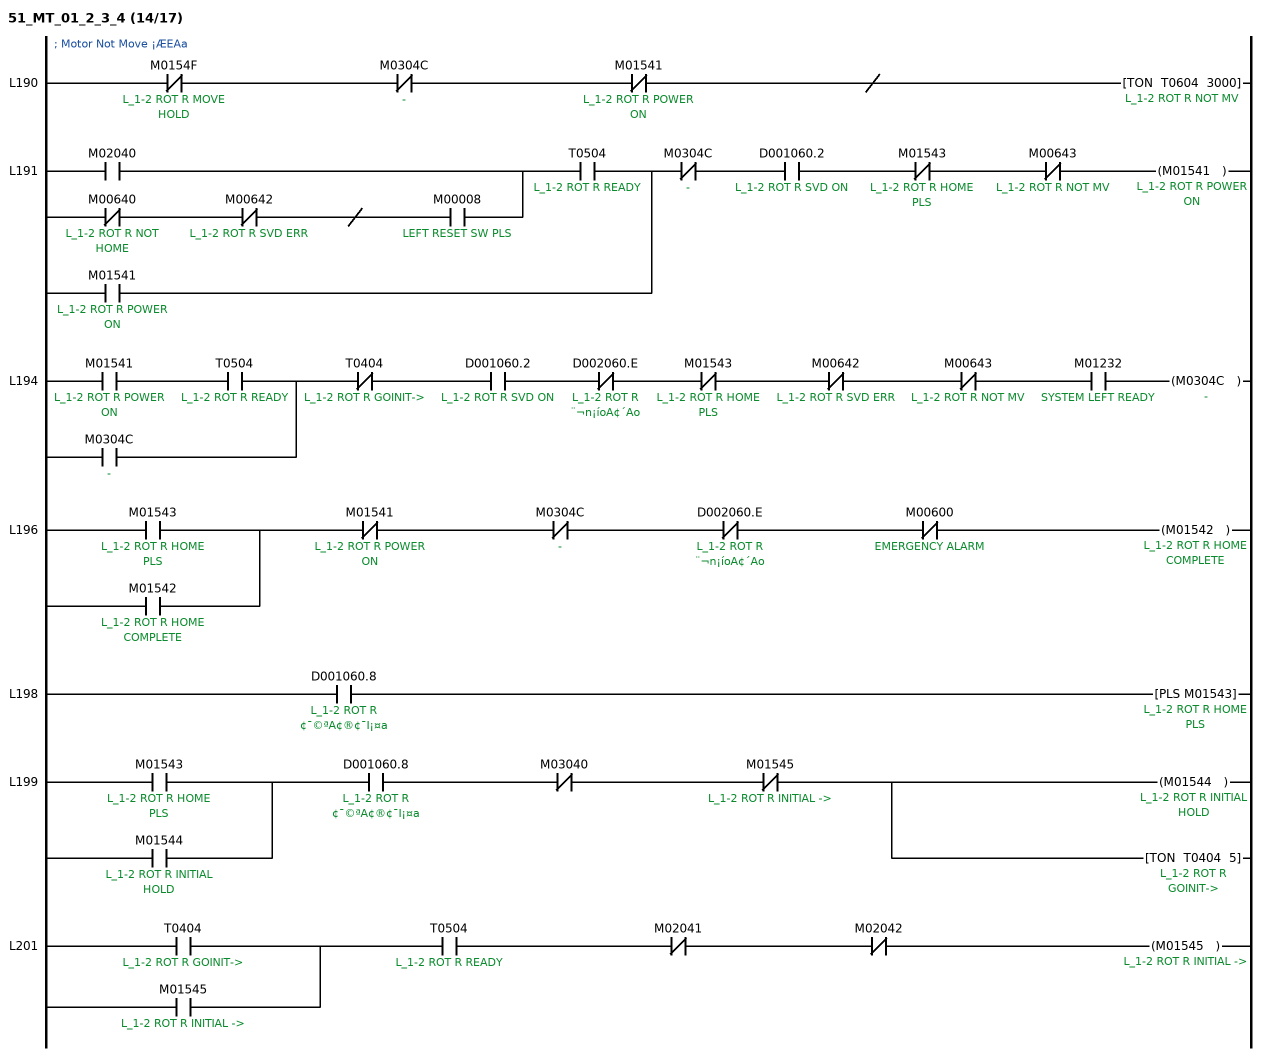
; L190
LOAD NOT  M0154F	// L_1-2 ROT R MOVE HOLD
AND NOT   M0304C	// -
AND NOT   M01541	// L_1-2 ROT R POWER ON
NOT
TON       T0604 3000	// L_1-2 ROT R NOT MV
// output comment: Motor Not Move ¡ÆEAa
; L191
LOAD      M02040
LOAD NOT  M00640	// L_1-2 ROT R NOT HOME
AND NOT   M00642	// L_1-2 ROT R SVD ERR
NOT
AND       M00008	// LEFT RESET SW PLS
OR LOAD
AND       T0504	// L_1-2 ROT R READY
OR        M01541	// L_1-2 ROT R POWER ON
AND NOT   M0304C	// -
AND       D001060.2	// L_1-2 ROT R SVD ON
AND NOT   M01543	// L_1-2 ROT R HOME PLS
AND NOT   M00643	// L_1-2 ROT R NOT MV
OUT       M01541	// L_1-2 ROT R POWER ON
; L194
LOAD      M01541	// L_1-2 ROT R POWER ON
AND       T0504	// L_1-2 ROT R READY
OR        M0304C	// -
AND NOT   T0404	// L_1-2 ROT R GOINIT->
AND       D001060.2	// L_1-2 ROT R SVD ON
AND NOT   D002060.E	// L_1-2 ROT R ¨¬n¡íoA¢´Ao
AND NOT   M01543	// L_1-2 ROT R HOME PLS
AND NOT   M00642	// L_1-2 ROT R SVD ERR
AND NOT   M00643	// L_1-2 ROT R NOT MV
AND       M01232	// SYSTEM LEFT READY
OUT       M0304C	// -
; L196
LOAD      M01543	// L_1-2 ROT R HOME PLS
OR        M01542	// L_1-2 ROT R HOME COMPLETE
AND NOT   M01541	// L_1-2 ROT R POWER ON
AND NOT   M0304C	// -
AND NOT   D002060.E	// L_1-2 ROT R ¨¬n¡íoA¢´Ao
AND NOT   M00600	// EMERGENCY ALARM
OUT       M01542	// L_1-2 ROT R HOME COMPLETE
; L198
LOAD      D001060.8	// L_1-2 ROT R ¢¯©ªA¢®¢¯I¡¤a
OUTP      M01543	// L_1-2 ROT R HOME PLS
; L199
LOAD      M01543	// L_1-2 ROT R HOME PLS
OR        M01544	// L_1-2 ROT R INITIAL HOLD
AND       D001060.8	// L_1-2 ROT R ¢¯©ªA¢®¢¯I¡¤a
AND NOT   M03040
AND NOT   M01545	// L_1-2 ROT R INITIAL ->
OUT       M01544	// L_1-2 ROT R INITIAL HOLD
TON       T0404 5	// L_1-2 ROT R GOINIT->
; L201
LOAD      T0404	// L_1-2 ROT R GOINIT->
OR        M01545	// L_1-2 ROT R INITIAL ->
AND       T0504	// L_1-2 ROT R READY
AND NOT   M02041
AND NOT   M02042
OUT       M01545	// L_1-2 ROT R INITIAL ->

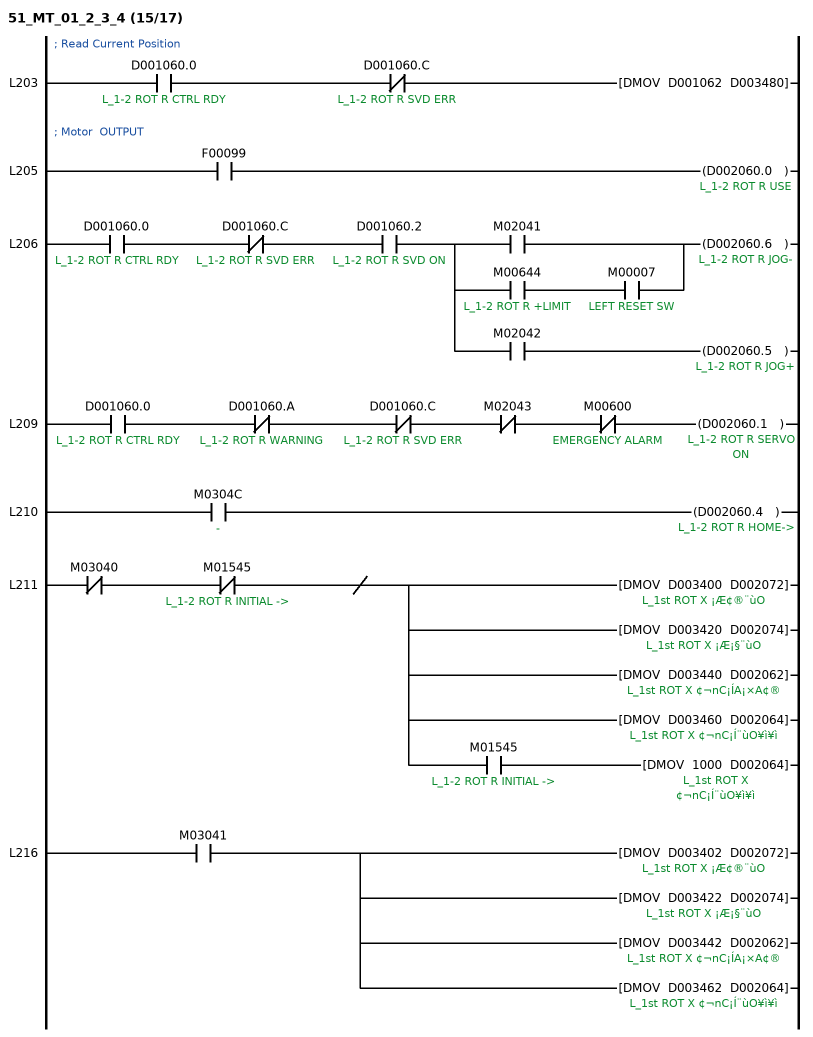
; L203
LOAD      D001060.0	// L_1-2 ROT R CTRL RDY
AND NOT   D001060.C	// L_1-2 ROT R SVD ERR
DMOV      D001062 D003480
// output comment: Read Current Position
//  Motor  OUTPUT
; L205
LOAD      F00099
OUT       D002060.0	// L_1-2 ROT R USE
; L206
LOAD      D001060.0	// L_1-2 ROT R CTRL RDY
AND NOT   D001060.C	// L_1-2 ROT R SVD ERR
AND       D001060.2	// L_1-2 ROT R SVD ON
MPUSH
LOAD      M02041
LOAD      M00644	// L_1-2 ROT R +LIMIT
AND       M00007	// LEFT RESET SW
OR LOAD
AND LOAD
OUT       D002060.6	// L_1-2 ROT R JOG-
MPOP
AND       M02042
OUT       D002060.5	// L_1-2 ROT R JOG+
; L209
LOAD      D001060.0	// L_1-2 ROT R CTRL RDY
AND NOT   D001060.A	// L_1-2 ROT R WARNING
AND NOT   D001060.C	// L_1-2 ROT R SVD ERR
AND NOT   M02043
AND NOT   M00600	// EMERGENCY ALARM
OUT       D002060.1	// L_1-2 ROT R SERVO ON
; L210
LOAD      M0304C	// -
OUT       D002060.4	// L_1-2 ROT R HOME->
; L211
LOAD NOT  M03040
AND NOT   M01545	// L_1-2 ROT R INITIAL ->
NOT
DMOV      D003400 D002072	// L_1st ROT X ¡Æ¢®¨ùO
DMOV      D003420 D002074	// L_1st ROT X ¡Æ¡§¨ùO
DMOV      D003440 D002062	// L_1st ROT X ¢¬nC¡ÍA¡×A¢®
DMOV      D003460 D002064	// L_1st ROT X ¢¬nC¡Í¨ùO¥ì¥ì
AND       M01545	// L_1-2 ROT R INITIAL ->
DMOV      1000 D002064	// L_1st ROT X ¢¬nC¡Í¨ùO¥ì¥ì
; L216
LOAD      M03041
DMOV      D003402 D002072	// L_1st ROT X ¡Æ¢®¨ùO
DMOV      D003422 D002074	// L_1st ROT X ¡Æ¡§¨ùO
DMOV      D003442 D002062	// L_1st ROT X ¢¬nC¡ÍA¡×A¢®
DMOV      D003462 D002064	// L_1st ROT X ¢¬nC¡Í¨ùO¥ì¥ì

